RoboDK station: kr30 cnc 070419 1.rdk

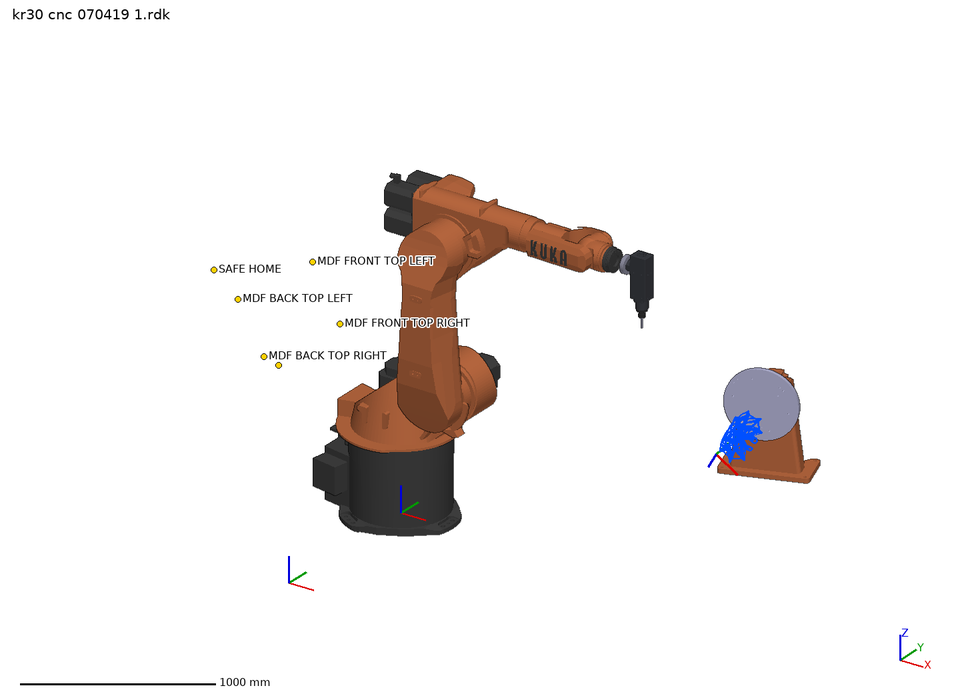
[picture v0: the station drawn from its stored meshes, robots at their saved joint values, targets as dots, program paths as lines]
Station kr30 cnc 070419 1. Poses are relative to the parent item; angles as X-Y-Z fixed-axis rotations.
  - frame GIGASHEEN 7th Axis Base at (0, 1000, 0) mm
    - robot KUKA KP1 MD250: 1 axes, payload 250 kg
        modified DH rows (alpha deg, a mm, theta deg, d mm): 0, 0, 0, 0
        base shift (1750, 1710, 820) mm, rotated rx 0 ry 90 rz -70 deg
        joint limits [-3600] to [3600]; home [0]; saved at [1487.65]
      - frame Reference Rhino at (0, -250, 250) mm
        - object RhinoPart at (0, 0, 0) mm
  - frame GIGASHEEN Base at (0, 2000, 0) mm
    - robot GIGASHEEN (model KUKA KR 30 HA): 6 axes, payload 30 kg, reach 2033 mm, repeatability 0.05 mm, weight 665 kg
        modified DH rows (alpha deg, a mm, theta deg, d mm): 0, 0, 0, 815; -90, 350, 0, 0; 0, 850, -90, 0; -90, 145, 0, 820; 90, 0, 0, 0; -90, 0, 180, 170
        joint limits [-185, -135, -120, -350, -119, -350] to [185, 35, 158, 350, 119, 350]; home [0, -90, 90, 0, 0, 0]; saved at [0, -90, 90, 0, 0, 0]
      - tool 1/2" End Mill TCP, TCP at (337.71, -2.2, 160.57) mm, rotated rx 0 ry 90 rz 0 deg, size 415.8 x 102 x 153.6 mm
    - target MDF BACK TOP LEFT (joint target) at (-335.18, -974.02, 1512.92) mm, rotated rx 85.17 ry 71.84 rz 47.05 deg; joints [27.716, -45.008, 102.25, 116.233, 75.695, -151.59, -681.46] of GIGASHEEN
    - target MDF FRONT TOP LEFT (joint target) at (-87.97, -665.25, 1668.52) mm, rotated rx 85.17 ry 71.84 rz 47.05 deg; joints [22.06, -21.631, 54.581, 104.768, 70.881, -126.376, -681.46] of GIGASHEEN
    - target MDF FRONT TOP RIGHT (joint target) at (4.03, -550.6, 1295.2) mm, rotated rx 85.17 ry 71.84 rz 47.05 deg; joints [10.053, -29.315, 70.245, 98.928, 81.917, -132.341, -681.46] of GIGASHEEN
    - target MDF BACK TOP RIGHT (joint target) at (-248.73, -867.72, 1165.36) mm, rotated rx 85.17 ry 71.84 rz 47.05 deg; joints [13.787, -50.344, 113.459, 104.66, 84.215, -154.683, -681.46] of GIGASHEEN
    - target MDF STOCK DEPTH (only use z axis value) (joint target) at (-166.67, -856.91, 1136.76) mm, rotated rx 85.17 ry 71.84 rz 47.05 deg; joints [11.502, -45.737, 110.222, 102.707, 85.519, -155.78, -681.46] of GIGASHEEN
    - target SAFE HOME (joint target) at (-1073.3, -134.71, 1136.76) mm, rotated rx 85.17 ry 71.84 rz 47.05 deg; joints [11.502, -69.45, 58.776, 88.861, 76.585, -79.989, -681.46] of GIGASHEEN
  - machining project RhinoPart Settings: rotZ(0) | rotX(90)*rotY(-155) | rotz(0)
  - program RhinoPart (1768 instructions, listed below)
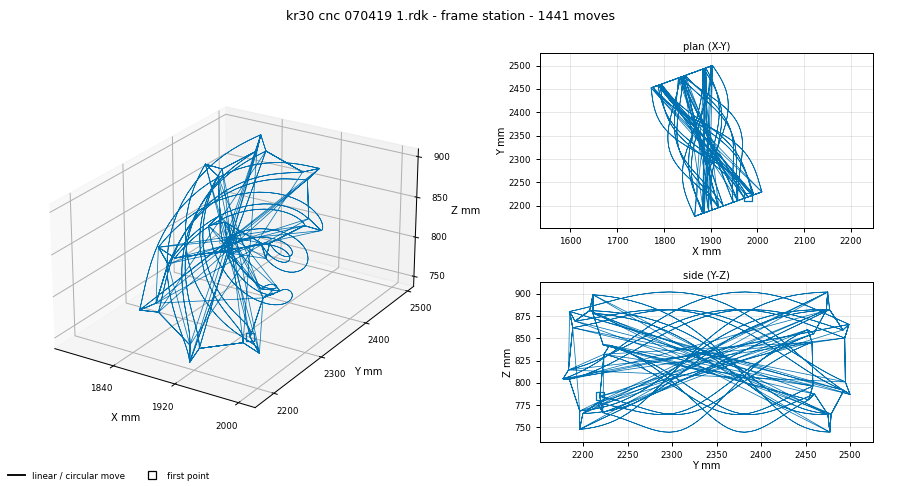
[picture p0: tool path of kr30 cnc 070419 1.rdk in frame station, 1441 of 1441 moves have a stored position in this frame; points joined in program order, loops and branches not executed]

--- program RhinoPart (robot GIGASHEEN) ---
  Set Ref.: Reference Rhino
  Set Tool: 1/2" End Mill TCP
  Show 1/2" End Mill TCP
  Set speed (1000.0 mm/s)
  MoveJ 1 to (58.93, 255.88, 290) mm, rotated rx -90 ry -25 rz 145.69 deg; joints [2.992, -45.858, 98.042, 40.619, -108.716, -6.951, -185.694]
  MoveL 2 to (58.93, 255.88, 290) mm, rotated rx -90 ry -25 rz 145.69 deg; joints [2.992, -45.858, 98.042, 40.619, -108.716, -6.951, -185.694]
  MoveL 3 to (58.93, 255.88, 290) mm, rotated rx -90 ry -25 rz 145.69 deg; joints [2.992, -45.858, 98.042, 40.619, -108.716, -6.951, -185.694]
  Set speed (60.0 mm/s)
  MoveL 4 to (37.11, 300.24, 290) mm, rotated rx -90 ry -25 rz -166.45 deg; joints [2.992, -46.004, 98.028, 40.584, -108.594, -7.061, -233.547]
  Set speed (1000.0 mm/s)
  MoveL 5 to (37.11, 300.24, 290) mm, rotated rx -90 ry -25 rz -166.45 deg; joints [2.992, -46.004, 98.028, 40.584, -108.594, -7.061, -233.547]
  Set speed (1000.0 mm/s)
  MoveL 6 to (-37.11, 208.63, 290) mm, rotated rx -90 ry -25 rz 8.11 deg; joints [2.992, -45.692, 98.056, 40.659, -108.852, -6.827, -408.107]
  MoveL 7 to (-37.11, 208.63, 290) mm, rotated rx -90 ry -25 rz 8.11 deg; joints [2.992, -45.692, 98.056, 40.659, -108.852, -6.827, -408.107]
  Set speed (60.0 mm/s)
  MoveL 8 to (-58.93, 252.99, 290) mm, rotated rx -90 ry -25 rz -42.9 deg; joints [2.992, -45.848, 98.043, 40.621, -108.724, -6.944, -357.096]
  Set speed (1000.0 mm/s)
  MoveL 9 to (-58.93, 252.99, 290) mm, rotated rx -90 ry -25 rz -42.9 deg; joints [2.992, -45.848, 98.043, 40.621, -108.724, -6.944, -357.096]
  Set speed (1000.0 mm/s)
  MoveL 10 to (21.11, 199.39, 290) mm, rotated rx -90 ry -25 rz 72.64 deg; joints [2.992, -45.658, 98.059, 40.667, -108.88, -6.802, -472.645]
  MoveL 11 to (21.11, 199.39, 290) mm, rotated rx -90 ry -25 rz 72.64 deg; joints [2.992, -45.658, 98.059, 40.667, -108.88, -6.802, -472.645]
  Set speed (60.0 mm/s)
  MoveL 12 to (34.79, 183.72, 290) mm, rotated rx -90 ry -25 rz 77.69 deg; joints [2.992, -46.56, 97.967, 40.451, -108.125, -7.483, -477.692]
  Set speed (1000.0 mm/s)
  MoveL 13 to (34.79, 183.72, 290) mm, rotated rx -90 ry -25 rz 77.69 deg; joints [2.992, -46.56, 97.967, 40.451, -108.125, -7.483, -477.692]
  Set speed (1000.0 mm/s)
  MoveL 14 to (21.11, 199.39, 290) mm, rotated rx -90 ry -25 rz 72.64 deg; joints [2.992, -45.658, 98.059, 40.667, -108.88, -6.802, -472.645]
  MoveL 15 to (21.11, 199.39, 290) mm, rotated rx -90 ry -25 rz 72.64 deg; joints [2.992, -45.658, 98.059, 40.667, -108.88, -6.802, -472.645]
  Set speed (60.0 mm/s)
  MoveL 16 to (-28.22, 202.67, 290) mm, rotated rx -90 ry -25 rz 19.2 deg; joints [2.992, -45.67, 98.058, 40.664, -108.87, -6.811, -419.196]
  Set speed (1000.0 mm/s)
  MoveL 17 to (-28.22, 202.67, 290) mm, rotated rx -90 ry -25 rz 19.2 deg; joints [2.992, -45.67, 98.058, 40.664, -108.87, -6.811, -419.196]
  Set speed (1000.0 mm/s)
  MoveL 18 to (-43.85, 188.95, 290) mm, rotated rx -90 ry -25 rz 14.31 deg; joints [2.992, -46.574, 97.966, 40.447, -108.114, -7.494, -414.314]
  MoveL 19 to (-43.85, 188.95, 290) mm, rotated rx -90 ry -25 rz 14.31 deg; joints [2.992, -46.574, 97.966, 40.447, -108.114, -7.494, -414.314]
  Set speed (60.0 mm/s)
  MoveL 20 to (-28.22, 202.67, 290) mm, rotated rx -90 ry -25 rz 19.2 deg; joints [2.992, -45.67, 98.058, 40.664, -108.87, -6.811, -419.196]
  Set speed (1000.0 mm/s)
  MoveL 21 to (-28.22, 202.67, 290) mm, rotated rx -90 ry -25 rz 19.2 deg; joints [2.992, -45.67, 98.058, 40.664, -108.87, -6.811, -419.196]
  Set speed (1000.0 mm/s)
  MoveL 22 to (-43.85, 188.95, 290) mm, rotated rx -90 ry -25 rz 14.31 deg; joints [2.992, -46.574, 97.966, 40.447, -108.114, -7.494, -414.314]
  MoveL 23 to (-43.85, 188.95, 290) mm, rotated rx -90 ry -25 rz 14.31 deg; joints [2.992, -46.574, 97.966, 40.447, -108.114, -7.494, -414.314]
  Set speed (60.0 mm/s)
  MoveL 24 to (-37.11, 208.63, 290) mm, rotated rx -90 ry -25 rz 8.11 deg; joints [2.992, -45.692, 98.056, 40.659, -108.852, -6.827, -408.107]
  Set speed (1000.0 mm/s)
  MoveL 25 to (-37.11, 208.63, 290) mm, rotated rx -90 ry -25 rz 8.11 deg; joints [2.992, -45.692, 98.056, 40.659, -108.852, -6.827, -408.107]
  Set speed (1000.0 mm/s)
  MoveL 26 to (-78.63, 259.66, 290) mm, rotated rx -90 ry -25 rz -47.01 deg; joints [2.992, -46.754, 97.943, 40.404, -107.959, -7.632, -352.994]
  MoveL 27 to (-78.63, 259.66, 290) mm, rotated rx -90 ry -25 rz -47.01 deg; joints [2.992, -46.754, 97.943, 40.404, -107.959, -7.632, -352.994]
  Set speed (60.0 mm/s)
  MoveL 28 to (-58.93, 252.99, 290) mm, rotated rx -90 ry -25 rz -42.9 deg; joints [2.992, -45.848, 98.043, 40.621, -108.724, -6.944, -357.096]
  Set speed (1000.0 mm/s)
  MoveL 29 to (-58.93, 252.99, 290) mm, rotated rx -90 ry -25 rz -42.9 deg; joints [2.992, -45.848, 98.043, 40.621, -108.724, -6.944, -357.096]
  Set speed (1000.0 mm/s)
  MoveL 30 to (-78.63, 259.66, 290) mm, rotated rx -90 ry -25 rz -47.01 deg; joints [2.992, -46.754, 97.943, 40.404, -107.959, -7.632, -352.994]
  MoveL 31 to (-78.63, 259.66, 290) mm, rotated rx -90 ry -25 rz -47.01 deg; joints [2.992, -46.754, 97.943, 40.404, -107.959, -7.632, -352.994]
  Set speed (60.0 mm/s)
  MoveL 32 to (-58.22, 263.67, 290) mm, rotated rx -90 ry -25 rz -53.21 deg; joints [2.992, -45.884, 98.039, 40.612, -108.694, -6.971, -346.787]
  Set speed (1000.0 mm/s)
  MoveL 33 to (-58.22, 263.67, 290) mm, rotated rx -90 ry -25 rz -53.21 deg; joints [2.992, -45.884, 98.039, 40.612, -108.694, -6.971, -346.787]
  Set speed (1000.0 mm/s)
  MoveL 34 to (-30.72, 304.75, 290) mm, rotated rx -90 ry -25 rz -100.71 deg; joints [2.992, -46.018, 98.027, 40.58, -108.582, -7.072, -299.294]
  MoveL 35 to (-30.72, 304.75, 290) mm, rotated rx -90 ry -25 rz -100.71 deg; joints [2.992, -46.018, 98.027, 40.58, -108.582, -7.072, -299.294]
  Set speed (60.0 mm/s)
  MoveL 36 to (-58.22, 263.67, 290) mm, rotated rx -90 ry -25 rz -53.21 deg; joints [2.992, -45.884, 98.039, 40.612, -108.694, -6.971, -346.787]
  Set speed (1000.0 mm/s)
  MoveL 37 to (-58.22, 263.67, 290) mm, rotated rx -90 ry -25 rz -53.21 deg; joints [2.992, -45.884, 98.039, 40.612, -108.694, -6.971, -346.787]
  Set speed (1000.0 mm/s)
  MoveL 38 to (-30.72, 304.75, 290) mm, rotated rx -90 ry -25 rz -100.71 deg; joints [2.992, -46.018, 98.027, 40.58, -108.582, -7.072, -299.294]
  MoveL 39 to (-30.72, 304.75, 290) mm, rotated rx -90 ry -25 rz -100.71 deg; joints [2.992, -46.018, 98.027, 40.58, -108.582, -7.072, -299.294]
  Set speed (60.0 mm/s)
  MoveL 40 to (-34.79, 325.15, 290) mm, rotated rx -90 ry -25 rz -105.16 deg; joints [2.992, -46.913, 97.922, 40.367, -107.822, -7.755, -294.84]
  Set speed (1000.0 mm/s)
  MoveL 41 to (-34.79, 325.15, 290) mm, rotated rx -90 ry -25 rz -105.16 deg; joints [2.992, -46.913, 97.922, 40.367, -107.822, -7.755, -294.84]
  Set speed (1000.0 mm/s)
  MoveL 42 to (-21.11, 309.47, 290) mm, rotated rx -90 ry -25 rz -110.46 deg; joints [2.992, -46.033, 98.025, 40.576, -108.57, -7.083, -289.544]
  MoveL 43 to (-21.11, 309.47, 290) mm, rotated rx -90 ry -25 rz -110.46 deg; joints [2.992, -46.033, 98.025, 40.576, -108.57, -7.083, -289.544]
  Set speed (60.0 mm/s)
  MoveL 44 to (-34.79, 325.15, 290) mm, rotated rx -90 ry -25 rz -105.16 deg; joints [2.992, -46.913, 97.922, 40.367, -107.822, -7.755, -294.84]
  Set speed (1000.0 mm/s)
  MoveL 45 to (-34.79, 325.15, 290) mm, rotated rx -90 ry -25 rz -105.16 deg; joints [2.992, -46.913, 97.922, 40.367, -107.822, -7.755, -294.84]
  Set speed (1000.0 mm/s)
  MoveL 46 to (-21.11, 309.47, 290) mm, rotated rx -90 ry -25 rz -110.46 deg; joints [2.992, -46.033, 98.025, 40.576, -108.57, -7.083, -289.544]
  MoveL 47 to (-21.11, 309.47, 290) mm, rotated rx -90 ry -25 rz -110.46 deg; joints [2.992, -46.033, 98.025, 40.576, -108.57, -7.083, -289.544]
  Set speed (60.0 mm/s)
  MoveL 48 to (28.22, 306.19, 290) mm, rotated rx -90 ry -25 rz -156.66 deg; joints [2.992, -46.023, 98.026, 40.579, -108.578, -7.075, -243.337]
  Set speed (1000.0 mm/s)
  MoveL 49 to (28.22, 306.19, 290) mm, rotated rx -90 ry -25 rz -156.66 deg; joints [2.992, -46.023, 98.026, 40.579, -108.578, -7.075, -243.337]
  Set speed (1000.0 mm/s)
  MoveL 50 to (43.85, 319.91, 290) mm, rotated rx -90 ry -25 rz -162.09 deg; joints [2.992, -46.901, 97.924, 40.37, -107.832, -7.745, -237.907]
  MoveL 51 to (43.85, 319.91, 290) mm, rotated rx -90 ry -25 rz -162.09 deg; joints [2.992, -46.901, 97.924, 40.37, -107.832, -7.745, -237.907]
  Set speed (60.0 mm/s)
  MoveL 52 to (28.22, 306.19, 290) mm, rotated rx -90 ry -25 rz -156.66 deg; joints [2.992, -46.023, 98.026, 40.579, -108.578, -7.075, -243.337]
  Set speed (1000.0 mm/s)
  MoveL 53 to (28.22, 306.19, 290) mm, rotated rx -90 ry -25 rz -156.66 deg; joints [2.992, -46.023, 98.026, 40.579, -108.578, -7.075, -243.337]
  Set speed (1000.0 mm/s)
  MoveL 54 to (43.85, 319.91, 290) mm, rotated rx -90 ry -25 rz -162.09 deg; joints [2.992, -46.901, 97.924, 40.37, -107.832, -7.745, -237.907]
  MoveL 55 to (43.85, 319.91, 290) mm, rotated rx -90 ry -25 rz -162.09 deg; joints [2.992, -46.901, 97.924, 40.37, -107.832, -7.745, -237.907]
  Set speed (60.0 mm/s)
  MoveL 56 to (37.11, 300.24, 290) mm, rotated rx -90 ry -25 rz -166.45 deg; joints [2.992, -46.004, 98.028, 40.584, -108.594, -7.061, -233.547]
  Set speed (1000.0 mm/s)
  MoveL 57 to (37.11, 300.24, 290) mm, rotated rx -90 ry -25 rz -166.45 deg; joints [2.992, -46.004, 98.028, 40.584, -108.594, -7.061, -233.547]
  Set speed (1000.0 mm/s)
  MoveL 58 to (78.63, 249.2, 290) mm, rotated rx -90 ry -25 rz 139.42 deg; joints [2.992, -46.728, 97.946, 40.411, -107.981, -7.612, -179.419]
  MoveL 59 to (78.63, 249.2, 290) mm, rotated rx -90 ry -25 rz 139.42 deg; joints [2.992, -46.728, 97.946, 40.411, -107.981, -7.612, -179.419]
  Set speed (60.0 mm/s)
  MoveL 60 to (58.93, 255.88, 290) mm, rotated rx -90 ry -25 rz 145.69 deg; joints [2.992, -45.858, 98.042, 40.619, -108.716, -6.951, -185.694]
  Set speed (1000.0 mm/s)
  MoveL 61 to (58.93, 255.88, 290) mm, rotated rx -90 ry -25 rz 145.69 deg; joints [2.992, -45.858, 98.042, 40.619, -108.716, -6.951, -185.694]
  Set speed (1000.0 mm/s)
  MoveL 62 to (78.63, 249.2, 290) mm, rotated rx -90 ry -25 rz 139.42 deg; joints [2.992, -46.728, 97.946, 40.411, -107.981, -7.612, -179.419]
  MoveL 63 to (78.63, 249.2, 290) mm, rotated rx -90 ry -25 rz 139.42 deg; joints [2.992, -46.728, 97.946, 40.411, -107.981, -7.612, -179.419]
  Set speed (60.0 mm/s)
  MoveL 64 to (58.22, 245.2, 290) mm, rotated rx -90 ry -25 rz 135.28 deg; joints [2.992, -45.821, 98.045, 40.627, -108.746, -6.924, -175.284]
  Set speed (1000.0 mm/s)
  MoveL 65 to (58.22, 245.2, 290) mm, rotated rx -90 ry -25 rz 135.28 deg; joints [2.992, -45.821, 98.045, 40.627, -108.746, -6.924, -175.284]
  Set speed (1000.0 mm/s)
  MoveL 66 to (30.72, 204.12, 290) mm, rotated rx -90 ry -25 rz 83.8 deg; joints [2.992, -45.676, 98.058, 40.663, -108.866, -6.815, -123.801]
  MoveL 67 to (30.72, 204.12, 290) mm, rotated rx -90 ry -25 rz 83.8 deg; joints [2.992, -45.676, 98.058, 40.663, -108.866, -6.815, -123.801]
  Set speed (60.0 mm/s)
  MoveL 68 to (58.22, 245.2, 290) mm, rotated rx -90 ry -25 rz 135.28 deg; joints [2.992, -45.821, 98.045, 40.627, -108.746, -6.924, -175.284]
  Set speed (1000.0 mm/s)
  MoveL 69 to (58.22, 245.2, 290) mm, rotated rx -90 ry -25 rz 135.28 deg; joints [2.992, -45.821, 98.045, 40.627, -108.746, -6.924, -175.284]
  Set speed (1000.0 mm/s)
  MoveL 70 to (30.72, 204.12, 290) mm, rotated rx -90 ry -25 rz 83.8 deg; joints [2.992, -45.676, 98.058, 40.663, -108.866, -6.815, -123.801]
  MoveL 71 to (30.72, 204.12, 290) mm, rotated rx -90 ry -25 rz 83.8 deg; joints [2.992, -45.676, 98.058, 40.663, -108.866, -6.815, -123.801]
  Set speed (60.0 mm/s)
  MoveL 72 to (34.79, 183.72, 290) mm, rotated rx -90 ry -25 rz 77.69 deg; joints [2.992, -46.56, 97.967, 40.451, -108.125, -7.483, -117.692]
  Set speed (1000.0 mm/s)
  MoveL 73 to (34.79, 183.72, 290) mm, rotated rx -90 ry -25 rz 77.69 deg; joints [2.992, -46.56, 97.967, 40.451, -108.125, -7.483, -117.692]
  Set speed (1000.0 mm/s)
  MoveL 74 to (-37.62, 299.82, 0) mm, rotated rx -90 ry -25 rz -92.94 deg; joints [-7.468, -50.311, 106.419, 34.538, -108.079, 0.675, 52.939]
  MoveL 75 to (-37.62, 299.82, 0) mm, rotated rx -90 ry -25 rz -92.94 deg; joints [-7.468, -50.311, 106.419, 34.538, -108.079, 0.675, 52.939]
  Set speed (60.0 mm/s)
  MoveL 76 to (10.16, 312.5, 0) mm, rotated rx -90 ry -25 rz -139.23 deg; joints [-7.468, -50.355, 106.415, 34.529, -108.039, 0.646, 99.233]
  Set speed (1000.0 mm/s)
  MoveL 77 to (10.16, 312.5, 0) mm, rotated rx -90 ry -25 rz -139.23 deg; joints [-7.468, -50.355, 106.415, 34.529, -108.039, 0.646, 99.233]
  Set speed (1000.0 mm/s)
  MoveL 78 to (-37.62, 299.82, 0) mm, rotated rx -90 ry -25 rz -92.94 deg; joints [-7.468, -50.311, 106.419, 34.538, -108.079, 0.675, 52.939]
  MoveL 79 to (-37.62, 299.82, 0) mm, rotated rx -90 ry -25 rz -92.94 deg; joints [-7.468, -50.311, 106.419, 34.538, -108.079, 0.675, 52.939]
  Set speed (60.0 mm/s)
  MoveL 80 to (-55.59, 310.29, 0) mm, rotated rx -90 ry -25 rz -87.32 deg; joints [-7.468, -51.259, 106.317, 34.349, -107.213, 0.052, 47.319]
  Set speed (1000.0 mm/s)
  MoveL 81 to (-55.59, 310.29, 0) mm, rotated rx -90 ry -25 rz -87.32 deg; joints [-7.468, -51.259, 106.317, 34.349, -107.213, 0.052, 47.319]
  Set speed (1000.0 mm/s)
  MoveL 82 to (-45.21, 292.27, 0) mm, rotated rx -90 ry -25 rz -83.07 deg; joints [-7.468, -50.285, 106.421, 34.543, -108.102, 0.692, 43.073]
  MoveL 83 to (-45.21, 292.27, 0) mm, rotated rx -90 ry -25 rz -83.07 deg; joints [-7.468, -50.285, 106.421, 34.543, -108.102, 0.692, 43.073]
  Set speed (60.0 mm/s)
  MoveL 84 to (-55.59, 310.29, 0) mm, rotated rx -90 ry -25 rz -87.32 deg; joints [-7.468, -51.259, 106.317, 34.349, -107.213, 0.052, 47.319]
  Set speed (1000.0 mm/s)
  MoveL 85 to (-55.59, 310.29, 0) mm, rotated rx -90 ry -25 rz -87.32 deg; joints [-7.468, -51.259, 106.317, 34.349, -107.213, 0.052, 47.319]
  Set speed (1000.0 mm/s)
  MoveL 86 to (-45.21, 292.27, 0) mm, rotated rx -90 ry -25 rz -83.07 deg; joints [-7.468, -50.285, 106.421, 34.543, -108.102, 0.692, 43.073]
  MoveL 87 to (-45.21, 292.27, 0) mm, rotated rx -90 ry -25 rz -83.07 deg; joints [-7.468, -50.285, 106.421, 34.543, -108.102, 0.692, 43.073]
  Set speed (60.0 mm/s)
  MoveL 88 to (-58.12, 244.54, 0) mm, rotated rx -90 ry -25 rz -34.64 deg; joints [-7.468, -50.113, 106.436, 34.578, -108.256, 0.804, -5.364]
  Set speed (1000.0 mm/s)
  MoveL 89 to (-58.12, 244.54, 0) mm, rotated rx -90 ry -25 rz -34.64 deg; joints [-7.468, -50.113, 106.436, 34.578, -108.256, 0.804, -5.364]
  Set speed (1000.0 mm/s)
  MoveL 90 to (-76.17, 234.21, 0) mm, rotated rx -90 ry -25 rz -28.29 deg; joints [-7.468, -51.057, 106.341, 34.389, -107.4, 0.186, -11.709]
  MoveL 91 to (-76.17, 234.21, 0) mm, rotated rx -90 ry -25 rz -28.29 deg; joints [-7.468, -51.057, 106.341, 34.389, -107.4, 0.186, -11.709]
  Set speed (60.0 mm/s)
  MoveL 92 to (-58.12, 244.54, 0) mm, rotated rx -90 ry -25 rz -34.64 deg; joints [-7.468, -50.113, 106.436, 34.578, -108.256, 0.804, -5.364]
  Set speed (1000.0 mm/s)
  MoveL 93 to (-58.12, 244.54, 0) mm, rotated rx -90 ry -25 rz -34.64 deg; joints [-7.468, -50.113, 106.436, 34.578, -108.256, 0.804, -5.364]
  Set speed (1000.0 mm/s)
  MoveL 94 to (-76.17, 234.21, 0) mm, rotated rx -90 ry -25 rz -28.29 deg; joints [-7.468, -51.057, 106.341, 34.389, -107.4, 0.186, -11.709]
  MoveL 95 to (-76.17, 234.21, 0) mm, rotated rx -90 ry -25 rz -28.29 deg; joints [-7.468, -51.057, 106.341, 34.389, -107.4, 0.186, -11.709]
  Set speed (60.0 mm/s)
  MoveL 96 to (-55.37, 234.2, 0) mm, rotated rx -90 ry -25 rz -24.07 deg; joints [-7.468, -50.074, 106.439, 34.586, -108.291, 0.829, -15.929]
  Set speed (1000.0 mm/s)
  MoveL 97 to (-55.37, 234.2, 0) mm, rotated rx -90 ry -25 rz -24.07 deg; joints [-7.468, -50.074, 106.439, 34.586, -108.291, 0.829, -15.929]
  Set speed (1000.0 mm/s)
  MoveL 98 to (-20.49, 199.16, 0) mm, rotated rx -90 ry -25 rz 28.05 deg; joints [-7.468, -49.938, 106.45, 34.613, -108.412, 0.917, -68.047]
  MoveL 99 to (-20.49, 199.16, 0) mm, rotated rx -90 ry -25 rz 28.05 deg; joints [-7.468, -49.938, 106.45, 34.613, -108.412, 0.917, -68.047]
  Set speed (60.0 mm/s)
  MoveL 100 to (-55.37, 234.2, 0) mm, rotated rx -90 ry -25 rz -24.07 deg; joints [-7.468, -50.074, 106.439, 34.586, -108.291, 0.829, -15.929]
  Set speed (1000.0 mm/s)
  MoveL 101 to (-55.37, 234.2, 0) mm, rotated rx -90 ry -25 rz -24.07 deg; joints [-7.468, -50.074, 106.439, 34.586, -108.291, 0.829, -15.929]
  Set speed (1000.0 mm/s)
  MoveL 102 to (-20.49, 199.16, 0) mm, rotated rx -90 ry -25 rz 28.05 deg; joints [-7.468, -49.938, 106.45, 34.613, -108.412, 0.917, -68.047]
  MoveL 103 to (-20.49, 199.16, 0) mm, rotated rx -90 ry -25 rz 28.05 deg; joints [-7.468, -49.938, 106.45, 34.613, -108.412, 0.917, -68.047]
  Set speed (60.0 mm/s)
  MoveL 104 to (-20.57, 178.36, 0) mm, rotated rx -90 ry -25 rz 33.98 deg; joints [-7.468, -50.9, 106.359, 34.42, -107.545, 0.29, -73.977]
  Set speed (1000.0 mm/s)
  MoveL 105 to (-20.57, 178.36, 0) mm, rotated rx -90 ry -25 rz 33.98 deg; joints [-7.468, -50.9, 106.359, 34.42, -107.545, 0.29, -73.977]
  Set speed (1000.0 mm/s)
  MoveL 106 to (-10.16, 196.36, 0) mm, rotated rx -90 ry -25 rz 39.27 deg; joints [-7.468, -49.927, 106.451, 34.616, -108.422, 0.924, -79.273]
  MoveL 107 to (-10.16, 196.36, 0) mm, rotated rx -90 ry -25 rz 39.27 deg; joints [-7.468, -49.927, 106.451, 34.616, -108.422, 0.924, -79.273]
  Set speed (60.0 mm/s)
  MoveL 108 to (-20.57, 178.36, 0) mm, rotated rx -90 ry -25 rz 33.98 deg; joints [-7.468, -50.9, 106.359, 34.42, -107.545, 0.29, -73.977]
  Set speed (1000.0 mm/s)
  MoveL 109 to (-20.57, 178.36, 0) mm, rotated rx -90 ry -25 rz 33.98 deg; joints [-7.468, -50.9, 106.359, 34.42, -107.545, 0.29, -73.977]
  Set speed (1000.0 mm/s)
  MoveL 110 to (-10.16, 196.36, 0) mm, rotated rx -90 ry -25 rz 39.27 deg; joints [-7.468, -49.927, 106.451, 34.616, -108.422, 0.924, -79.273]
  MoveL 111 to (-10.16, 196.36, 0) mm, rotated rx -90 ry -25 rz 39.27 deg; joints [-7.468, -49.927, 106.451, 34.616, -108.422, 0.924, -79.273]
  Set speed (60.0 mm/s)
  MoveL 112 to (37.62, 209.05, 0) mm, rotated rx -90 ry -25 rz 92.57 deg; joints [-7.468, -49.977, 106.447, 34.605, -108.377, 0.891, -132.574]
  Set speed (1000.0 mm/s)
  MoveL 113 to (37.62, 209.05, 0) mm, rotated rx -90 ry -25 rz 92.57 deg; joints [-7.468, -49.977, 106.447, 34.605, -108.377, 0.891, -132.574]
  Set speed (1000.0 mm/s)
  MoveL 114 to (55.59, 198.58, 0) mm, rotated rx -90 ry -25 rz 97.23 deg; joints [-7.468, -50.957, 106.353, 34.408, -107.492, 0.252, -137.234]
  MoveL 115 to (55.59, 198.58, 0) mm, rotated rx -90 ry -25 rz 97.23 deg; joints [-7.468, -50.957, 106.353, 34.408, -107.492, 0.252, -137.234]
  Set speed (60.0 mm/s)
  MoveL 116 to (37.62, 209.05, 0) mm, rotated rx -90 ry -25 rz 92.57 deg; joints [-7.468, -49.977, 106.447, 34.605, -108.377, 0.891, -132.574]
  Set speed (1000.0 mm/s)
  MoveL 117 to (37.62, 209.05, 0) mm, rotated rx -90 ry -25 rz 92.57 deg; joints [-7.468, -49.977, 106.447, 34.605, -108.377, 0.891, -132.574]
  Set speed (1000.0 mm/s)
  MoveL 118 to (55.59, 198.58, 0) mm, rotated rx -90 ry -25 rz 97.23 deg; joints [-7.468, -50.957, 106.353, 34.408, -107.492, 0.252, -137.234]
  MoveL 119 to (55.59, 198.58, 0) mm, rotated rx -90 ry -25 rz 97.23 deg; joints [-7.468, -50.957, 106.353, 34.408, -107.492, 0.252, -137.234]
  Set speed (60.0 mm/s)
  MoveL 120 to (45.21, 216.6, 0) mm, rotated rx -90 ry -25 rz 103.54 deg; joints [-7.468, -50.007, 106.445, 34.599, -108.351, 0.872, -143.543]
  Set speed (1000.0 mm/s)
  MoveL 121 to (45.21, 216.6, 0) mm, rotated rx -90 ry -25 rz 103.54 deg; joints [-7.468, -50.007, 106.445, 34.599, -108.351, 0.872, -143.543]
  Set speed (1000.0 mm/s)
  MoveL 122 to (58.12, 264.32, 0) mm, rotated rx -90 ry -25 rz 153.85 deg; joints [-7.468, -50.186, 106.43, 34.563, -108.191, 0.757, -193.845]
  MoveL 123 to (58.12, 264.32, 0) mm, rotated rx -90 ry -25 rz 153.85 deg; joints [-7.468, -50.186, 106.43, 34.563, -108.191, 0.757, -193.845]
  Set speed (60.0 mm/s)
  MoveL 124 to (45.21, 216.6, 0) mm, rotated rx -90 ry -25 rz 103.54 deg; joints [-7.468, -50.007, 106.445, 34.599, -108.351, 0.872, -143.543]
  Set speed (1000.0 mm/s)
  MoveL 125 to (45.21, 216.6, 0) mm, rotated rx -90 ry -25 rz 103.54 deg; joints [-7.468, -50.007, 106.445, 34.599, -108.351, 0.872, -143.543]
  Set speed (1000.0 mm/s)
  MoveL 126 to (58.12, 264.32, 0) mm, rotated rx -90 ry -25 rz 153.85 deg; joints [-7.468, -50.186, 106.43, 34.563, -108.191, 0.757, -193.845]
  MoveL 127 to (58.12, 264.32, 0) mm, rotated rx -90 ry -25 rz 153.85 deg; joints [-7.468, -50.186, 106.43, 34.563, -108.191, 0.757, -193.845]
  Set speed (60.0 mm/s)
  MoveL 128 to (76.17, 274.65, 0) mm, rotated rx -90 ry -25 rz 157.93 deg; joints [-7.468, -51.166, 106.328, 34.367, -107.299, 0.114, -197.935]
  Set speed (1000.0 mm/s)
  MoveL 129 to (76.17, 274.65, 0) mm, rotated rx -90 ry -25 rz 157.93 deg; joints [-7.468, -51.166, 106.328, 34.367, -107.299, 0.114, -197.935]
  Set speed (1000.0 mm/s)
  MoveL 130 to (55.37, 274.67, 0) mm, rotated rx -90 ry -25 rz 164.01 deg; joints [-7.468, -50.223, 106.427, 34.556, -108.158, 0.732, -204.014]
  MoveL 131 to (55.37, 274.67, 0) mm, rotated rx -90 ry -25 rz 164.01 deg; joints [-7.468, -50.223, 106.427, 34.556, -108.158, 0.732, -204.014]
  Set speed (60.0 mm/s)
  MoveL 132 to (76.17, 274.65, 0) mm, rotated rx -90 ry -25 rz 157.93 deg; joints [-7.468, -51.166, 106.328, 34.367, -107.299, 0.114, -197.935]
  Set speed (1000.0 mm/s)
  MoveL 133 to (76.17, 274.65, 0) mm, rotated rx -90 ry -25 rz 157.93 deg; joints [-7.468, -51.166, 106.328, 34.367, -107.299, 0.114, -197.935]
  Set speed (1000.0 mm/s)
  MoveL 134 to (55.37, 274.67, 0) mm, rotated rx -90 ry -25 rz 164.01 deg; joints [-7.468, -50.223, 106.427, 34.556, -108.158, 0.732, -204.014]
  MoveL 135 to (55.37, 274.67, 0) mm, rotated rx -90 ry -25 rz 164.01 deg; joints [-7.468, -50.223, 106.427, 34.556, -108.158, 0.732, -204.014]
  Set speed (60.0 mm/s)
  MoveL 136 to (20.49, 309.71, 0) mm, rotated rx -90 ry -25 rz -148.94 deg; joints [-7.468, -50.346, 106.416, 34.531, -108.048, 0.653, -251.057]
  Set speed (1000.0 mm/s)
  MoveL 137 to (20.49, 309.71, 0) mm, rotated rx -90 ry -25 rz -148.94 deg; joints [-7.468, -50.346, 106.416, 34.531, -108.048, 0.653, -251.057]
  Set speed (1000.0 mm/s)
  MoveL 138 to (20.57, 330.51, 0) mm, rotated rx -90 ry -25 rz -144.34 deg; joints [-7.468, -51.311, 106.31, 34.338, -107.164, 0.017, -255.665]
  MoveL 139 to (20.57, 330.51, 0) mm, rotated rx -90 ry -25 rz -144.34 deg; joints [-7.468, -51.311, 106.31, 34.338, -107.164, 0.017, -255.665]
  Set speed (60.0 mm/s)
  MoveL 140 to (20.49, 309.71, 0) mm, rotated rx -90 ry -25 rz -148.94 deg; joints [-7.468, -50.346, 106.416, 34.531, -108.048, 0.653, -251.057]
  Set speed (1000.0 mm/s)
  MoveL 141 to (20.49, 309.71, 0) mm, rotated rx -90 ry -25 rz -148.94 deg; joints [-7.468, -50.346, 106.416, 34.531, -108.048, 0.653, -251.057]
  Set speed (1000.0 mm/s)
  MoveL 142 to (20.57, 330.51, 0) mm, rotated rx -90 ry -25 rz -144.34 deg; joints [-7.468, -51.311, 106.31, 34.338, -107.164, 0.017, -255.665]
  MoveL 143 to (20.57, 330.51, 0) mm, rotated rx -90 ry -25 rz -144.34 deg; joints [-7.468, -51.311, 106.31, 34.338, -107.164, 0.017, -255.665]
  Set speed (60.0 mm/s)
  MoveL 144 to (10.16, 312.5, 0) mm, rotated rx -90 ry -25 rz -139.23 deg; joints [-7.468, -50.355, 106.415, 34.529, -108.039, 0.646, -260.767]
  Set speed (1000.0 mm/s)
  MoveL 145 to (10.16, 312.5, 0) mm, rotated rx -90 ry -25 rz -139.23 deg; joints [-7.468, -50.355, 106.415, 34.529, -108.039, 0.646, -260.767]
  Set speed (1000.0 mm/s)
  MoveL 146 to (-37.62, 299.82, 0) mm, rotated rx -90 ry -25 rz -92.94 deg; joints [-7.468, -50.311, 106.419, 34.538, -108.079, 0.675, -307.061]
  MoveL 147 to (-37.62, 299.82, 0) mm, rotated rx -90 ry -25 rz -92.94 deg; joints [-7.468, -50.311, 106.419, 34.538, -108.079, 0.675, -307.061]
  Set speed (60.0 mm/s)
  MoveL 148 to (-40.85, 296.93, 10) mm, rotated rx -90 ry -25 rz -88.96 deg; joints [-7.088, -50.198, 106.219, 34.78, -108.128, 0.44, -311.039]
  MoveL 149 to (-44.15, 293.5, 20) mm, rotated rx -90 ry -25 rz -84.58 deg; joints [-6.709, -50.079, 106.012, 35.02, -108.177, 0.204, -315.425]
  MoveL 150 to (-47.39, 289.5, 30) mm, rotated rx -90 ry -25 rz -79.81 deg; joints [-6.332, -49.955, 105.8, 35.259, -108.227, -0.032, -320.19]
  MoveL 151 to (-50.45, 284.92, 40) mm, rotated rx -90 ry -25 rz -74.69 deg; joints [-5.956, -49.826, 105.582, 35.496, -108.277, -0.268, -325.308]
  MoveL 152 to (-53.21, 279.8, 50) mm, rotated rx -90 ry -25 rz -69.25 deg; joints [-5.581, -49.692, 105.357, 35.732, -108.326, -0.504, -330.751]
  MoveL 153 to (-55.55, 274.16, 60) mm, rotated rx -90 ry -25 rz -63.51 deg; joints [-5.207, -49.552, 105.127, 35.966, -108.376, -0.74, -336.493]
  MoveL 154 to (-57.35, 268.08, 70) mm, rotated rx -90 ry -25 rz -57.49 deg; joints [-4.834, -49.408, 104.89, 36.198, -108.425, -0.977, -342.507]
  MoveL 155 to (-58.51, 261.62, 80) mm, rotated rx -90 ry -25 rz -51.24 deg; joints [-4.463, -49.259, 104.647, 36.429, -108.474, -1.215, -348.765]
  MoveL 156 to (-58.95, 254.91, 90) mm, rotated rx -90 ry -25 rz -44.76 deg; joints [-4.093, -49.106, 104.398, 36.657, -108.522, -1.454, -355.24]
  MoveL 157 to (-58.6, 248.05, 100) mm, rotated rx -90 ry -25 rz -38.1 deg; joints [-3.725, -48.95, 104.143, 36.884, -108.569, -1.693, -361.902]
  MoveL 158 to (-57.44, 241.19, 110) mm, rotated rx -90 ry -25 rz -31.28 deg; joints [-3.358, -48.79, 103.881, 37.108, -108.614, -1.935, -368.721]
  MoveL 159 to (-55.46, 234.45, 120) mm, rotated rx -90 ry -25 rz -24.34 deg; joints [-2.992, -48.627, 103.613, 37.33, -108.658, -2.178, -375.664]
  MoveL 160 to (-52.68, 227.97, 130) mm, rotated rx -90 ry -25 rz -17.3 deg; joints [-2.628, -48.462, 103.339, 37.55, -108.698, -2.423, -382.696]
  MoveL 161 to (-49.15, 221.88, 140) mm, rotated rx -90 ry -25 rz -10.22 deg; joints [-2.265, -48.294, 103.059, 37.767, -108.736, -2.671, -389.78]
  MoveL 162 to (-44.94, 216.28, 150) mm, rotated rx -90 ry -25 rz -3.12 deg; joints [-1.904, -48.126, 102.771, 37.981, -108.771, -2.922, -396.877]
  MoveL 163 to (-40.17, 211.29, 160) mm, rotated rx -90 ry -25 rz 3.94 deg; joints [-1.544, -47.956, 102.478, 38.192, -108.802, -3.176, -403.944]
  MoveL 164 to (-34.94, 206.95, 170) mm, rotated rx -90 ry -25 rz 10.94 deg; joints [-1.185, -47.786, 102.178, 38.401, -108.829, -3.434, -410.939]
  MoveL 165 to (-29.38, 203.32, 180) mm, rotated rx -90 ry -25 rz 17.81 deg; joints [-0.828, -47.615, 101.871, 38.606, -108.852, -3.696, -417.814]
  MoveL 166 to (-23.62, 200.42, 190) mm, rotated rx -90 ry -25 rz 24.52 deg; joints [-0.473, -47.444, 101.557, 38.809, -108.871, -3.961, -424.525]
  MoveL 167 to (-17.8, 198.23, 200) mm, rotated rx -90 ry -25 rz 31.02 deg; joints [-0.119, -47.272, 101.237, 39.008, -108.886, -4.23, -431.023]
  MoveL 168 to (-12.04, 196.73, 210) mm, rotated rx -90 ry -25 rz 37.26 deg; joints [0.233, -47.1, 100.911, 39.204, -108.897, -4.503, -437.262]
  MoveL 169 to (-6.46, 195.84, 220) mm, rotated rx -90 ry -25 rz 43.2 deg; joints [0.584, -46.927, 100.577, 39.397, -108.905, -4.78, -443.197]
  MoveL 170 to (-1.16, 195.49, 230) mm, rotated rx -90 ry -25 rz 48.78 deg; joints [0.933, -46.752, 100.237, 39.587, -108.909, -5.06, -448.782]
  MoveL 171 to (3.78, 195.6, 240) mm, rotated rx -90 ry -25 rz 53.97 deg; joints [1.28, -46.576, 99.891, 39.774, -108.91, -5.344, -453.974]
  MoveL 172 to (8.28, 196.07, 250) mm, rotated rx -90 ry -25 rz 58.73 deg; joints [1.626, -46.398, 99.538, 39.958, -108.908, -5.631, -458.733]
  MoveL 173 to (12.3, 196.78, 260) mm, rotated rx -90 ry -25 rz 63.02 deg; joints [1.97, -46.218, 99.178, 40.139, -108.904, -5.92, -463.017]
  MoveL 174 to (15.8, 197.64, 270) mm, rotated rx -90 ry -25 rz 66.79 deg; joints [2.312, -46.035, 98.812, 40.318, -108.898, -6.212, -466.788]
  MoveL 175 to (18.74, 198.54, 280) mm, rotated rx -90 ry -25 rz 70.01 deg; joints [2.653, -45.848, 98.439, 40.494, -108.89, -6.506, -470.01]
  MoveL 176 to (21.11, 199.39, 290) mm, rotated rx -90 ry -25 rz 72.64 deg; joints [2.992, -45.658, 98.059, 40.667, -108.88, -6.802, -472.645]
  Set speed (1000.0 mm/s)
  MoveL 177 to (21.11, 199.39, 290) mm, rotated rx -90 ry -25 rz 72.64 deg; joints [2.992, -45.658, 98.059, 40.667, -108.88, -6.802, -472.645]
  Set speed (1000.0 mm/s)
  MoveL 178 to (10.16, 312.5, 0) mm, rotated rx -90 ry -25 rz -139.23 deg; joints [-7.468, -50.355, 106.415, 34.529, -108.039, 0.646, -620.767]
  MoveL 179 to (10.16, 312.5, 0) mm, rotated rx -90 ry -25 rz -139.23 deg; joints [-7.468, -50.355, 106.415, 34.529, -108.039, 0.646, -620.767]
  Set speed (60.0 mm/s)
  MoveL 180 to (-37.62, 299.82, 0) mm, rotated rx -90 ry -25 rz -92.94 deg; joints [-7.468, -50.311, 106.419, 34.538, -108.079, 0.675, -667.061]
  Set speed (1000.0 mm/s)
  MoveL 181 to (-37.62, 299.82, 0) mm, rotated rx -90 ry -25 rz -92.94 deg; joints [-7.468, -50.311, 106.419, 34.538, -108.079, 0.675, -667.061]
  Set speed (1000.0 mm/s)
  MoveL 182 to (-28.22, 202.67, 290) mm, rotated rx -90 ry -25 rz 19.2 deg; joints [2.992, -45.67, 98.058, 40.664, -108.87, -6.811, -779.196]
  MoveL 183 to (-28.22, 202.67, 290) mm, rotated rx -90 ry -25 rz 19.2 deg; joints [2.992, -45.67, 98.058, 40.664, -108.87, -6.811, -779.196]
  Set speed (60.0 mm/s)
  MoveL 184 to (21.11, 199.39, 290) mm, rotated rx -90 ry -25 rz 72.64 deg; joints [2.992, -45.658, 98.059, 40.667, -108.88, -6.802, -832.645]
  Set speed (1000.0 mm/s)
  MoveL 185 to (21.11, 199.39, 290) mm, rotated rx -90 ry -25 rz 72.64 deg; joints [2.992, -45.658, 98.059, 40.667, -108.88, -6.802, -832.645]
  Set speed (1000.0 mm/s)
  MoveL 186 to (-28.22, 202.67, 290) mm, rotated rx -90 ry -25 rz 19.2 deg; joints [2.992, -45.67, 98.058, 40.664, -108.87, -6.811, -779.196]
  MoveL 187 to (-28.22, 202.67, 290) mm, rotated rx -90 ry -25 rz 19.2 deg; joints [2.992, -45.67, 98.058, 40.664, -108.87, -6.811, -779.196]
  Set speed (60.0 mm/s)
  MoveL 188 to (-30.4, 203.93, 280) mm, rotated rx -90 ry -25 rz 16.58 deg; joints [2.653, -45.868, 98.437, 40.489, -108.873, -6.521, -776.579]
  MoveL 189 to (-33, 205.58, 270) mm, rotated rx -90 ry -25 rz 13.39 deg; joints [2.312, -46.064, 98.809, 40.311, -108.874, -6.234, -773.391]
  MoveL 190 to (-35.92, 207.69, 260) mm, rotated rx -90 ry -25 rz 9.67 deg; joints [1.97, -46.258, 99.175, 40.13, -108.871, -5.95, -769.674]
  MoveL 191 to (-39.07, 210.28, 250) mm, rotated rx -90 ry -25 rz 5.47 deg; joints [1.626, -46.451, 99.533, 39.946, -108.865, -5.669, -765.473]
  MoveL 192 to (-42.34, 213.41, 240) mm, rotated rx -90 ry -25 rz 0.83 deg; joints [1.28, -46.642, 99.885, 39.758, -108.855, -5.392, -760.831]
  MoveL 193 to (-45.62, 217.1, 230) mm, rotated rx -90 ry -25 rz -4.21 deg; joints [0.933, -46.832, 100.231, 39.568, -108.842, -5.119, -755.794]
  MoveL 194 to (-48.8, 221.36, 220) mm, rotated rx -90 ry -25 rz -9.59 deg; joints [0.584, -47.021, 100.57, 39.375, -108.826, -4.849, -750.406]
  MoveL 195 to (-51.74, 226.19, 210) mm, rotated rx -90 ry -25 rz -15.29 deg; joints [0.233, -47.209, 100.902, 39.178, -108.806, -4.582, -744.713]
  MoveL 196 to (-54.33, 231.55, 200) mm, rotated rx -90 ry -25 rz -21.24 deg; joints [-0.119, -47.395, 101.227, 38.979, -108.783, -4.319, -738.758]
  MoveL 197 to (-56.44, 237.4, 190) mm, rotated rx -90 ry -25 rz -27.41 deg; joints [-0.473, -47.58, 101.546, 38.777, -108.756, -4.059, -732.587]
  MoveL 198 to (-57.96, 243.66, 180) mm, rotated rx -90 ry -25 rz -33.76 deg; joints [-0.828, -47.763, 101.858, 38.572, -108.727, -3.801, -726.24]
  MoveL 199 to (-58.8, 250.25, 170) mm, rotated rx -90 ry -25 rz -40.24 deg; joints [-1.185, -47.944, 102.164, 38.365, -108.694, -3.547, -719.76]
  MoveL 200 to (-58.89, 257.04, 160) mm, rotated rx -90 ry -25 rz -46.82 deg; joints [-1.544, -48.123, 102.464, 38.154, -108.66, -3.294, -713.183]
  MoveL 201 to (-58.18, 263.92, 150) mm, rotated rx -90 ry -25 rz -53.45 deg; joints [-1.904, -48.298, 102.757, 37.942, -108.623, -3.043, -706.549]
  MoveL 202 to (-56.65, 270.74, 140) mm, rotated rx -90 ry -25 rz -60.11 deg; joints [-2.265, -48.47, 103.043, 37.727, -108.585, -2.794, -699.89]
  MoveL 203 to (-54.3, 277.38, 130) mm, rotated rx -90 ry -25 rz -66.76 deg; joints [-2.628, -48.638, 103.324, 37.51, -108.546, -2.546, -693.241]
  MoveL 204 to (-51.17, 283.7, 120) mm, rotated rx -90 ry -25 rz -73.37 deg; joints [-2.992, -48.802, 103.598, 37.291, -108.506, -2.299, -686.632]
  MoveL 205 to (-47.33, 289.58, 110) mm, rotated rx -90 ry -25 rz -79.91 deg; joints [-3.358, -48.961, 103.866, 37.07, -108.466, -2.053, -680.094]
  MoveL 206 to (-42.85, 294.92, 100) mm, rotated rx -90 ry -25 rz -86.35 deg; joints [-3.725, -49.114, 104.128, 36.848, -108.426, -1.807, -673.654]
  MoveL 207 to (-37.86, 299.62, 90) mm, rotated rx -90 ry -25 rz -92.66 deg; joints [-4.093, -49.263, 104.384, 36.623, -108.386, -1.561, -667.341]
  MoveL 208 to (-32.46, 303.64, 80) mm, rotated rx -90 ry -25 rz -98.82 deg; joints [-4.463, -49.406, 104.634, 36.397, -108.346, -1.315, -661.181]
  MoveL 209 to (-26.8, 306.94, 70) mm, rotated rx -90 ry -25 rz -104.8 deg; joints [-4.834, -49.543, 104.878, 36.169, -108.307, -1.069, -655.202]
  MoveL 210 to (-21, 309.52, 60) mm, rotated rx -90 ry -25 rz -110.57 deg; joints [-5.207, -49.675, 105.115, 35.94, -108.268, -0.823, -649.431]
  MoveL 211 to (-15.19, 311.39, 50) mm, rotated rx -90 ry -25 rz -116.1 deg; joints [-5.581, -49.801, 105.347, 35.709, -108.23, -0.577, -643.896]
  MoveL 212 to (-9.5, 312.61, 40) mm, rotated rx -90 ry -25 rz -121.38 deg; joints [-5.956, -49.921, 105.573, 35.476, -108.192, -0.331, -638.624]
  MoveL 213 to (-4.03, 313.25, 30) mm, rotated rx -90 ry -25 rz -126.35 deg; joints [-6.332, -50.037, 105.793, 35.242, -108.154, -0.086, -633.645]
  MoveL 214 to (1.12, 313.37, 20) mm, rotated rx -90 ry -25 rz -131.01 deg; joints [-6.709, -50.147, 106.006, 35.006, -108.116, 0.159, -628.989]
  MoveL 215 to (5.87, 313.09, 10) mm, rotated rx -90 ry -25 rz -135.31 deg; joints [-7.088, -50.253, 106.214, 34.768, -108.078, 0.403, -624.685]
  MoveL 216 to (10.16, 312.5, 0) mm, rotated rx -90 ry -25 rz -139.23 deg; joints [-7.468, -50.355, 106.415, 34.529, -108.039, 0.646, -620.767]
  Set speed (1000.0 mm/s)
  MoveL 217 to (10.16, 312.5, 0) mm, rotated rx -90 ry -25 rz -139.23 deg; joints [-7.468, -50.355, 106.415, 34.529, -108.039, 0.646, -620.767]
  Set speed (1000.0 mm/s)
  MoveL 218 to (-37.62, 299.82, 0) mm, rotated rx -90 ry -25 rz -92.94 deg; joints [-7.468, -50.311, 106.419, 34.538, -108.079, 0.675, -667.061]
  MoveL 219 to (-37.62, 299.82, 0) mm, rotated rx -90 ry -25 rz -92.94 deg; joints [-7.468, -50.311, 106.419, 34.538, -108.079, 0.675, -667.061]
  Set speed (60.0 mm/s)
  MoveL 220 to (-40.85, 296.93, 10) mm, rotated rx -90 ry -25 rz -88.96 deg; joints [-7.088, -50.198, 106.219, 34.78, -108.128, 0.44, -671.039]
  MoveL 221 to (-44.15, 293.5, 20) mm, rotated rx -90 ry -25 rz -84.58 deg; joints [-6.709, -50.079, 106.012, 35.02, -108.177, 0.204, -675.425]
  MoveL 222 to (-47.39, 289.5, 30) mm, rotated rx -90 ry -25 rz -79.81 deg; joints [-6.332, -49.955, 105.8, 35.259, -108.227, -0.032, -680.19]
  MoveL 223 to (-50.45, 284.92, 40) mm, rotated rx -90 ry -25 rz -74.69 deg; joints [-5.956, -49.826, 105.582, 35.496, -108.277, -0.268, -685.308]
  MoveL 224 to (-53.21, 279.8, 50) mm, rotated rx -90 ry -25 rz -69.25 deg; joints [-5.581, -49.692, 105.357, 35.732, -108.326, -0.504, -690.751]
  MoveL 225 to (-55.55, 274.16, 60) mm, rotated rx -90 ry -25 rz -63.51 deg; joints [-5.207, -49.552, 105.127, 35.966, -108.376, -0.74, -696.493]
  MoveL 226 to (-57.35, 268.08, 70) mm, rotated rx -90 ry -25 rz -57.49 deg; joints [-4.834, -49.408, 104.89, 36.198, -108.425, -0.977, -702.507]
  MoveL 227 to (-58.51, 261.62, 80) mm, rotated rx -90 ry -25 rz -51.24 deg; joints [-4.463, -49.259, 104.647, 36.429, -108.474, -1.215, -708.765]
  MoveL 228 to (-58.95, 254.91, 90) mm, rotated rx -90 ry -25 rz -44.76 deg; joints [-4.093, -49.106, 104.398, 36.657, -108.522, -1.454, -715.24]
  MoveL 229 to (-58.6, 248.05, 100) mm, rotated rx -90 ry -25 rz -38.1 deg; joints [-3.725, -48.95, 104.143, 36.884, -108.569, -1.693, -721.902]
  MoveL 230 to (-57.44, 241.19, 110) mm, rotated rx -90 ry -25 rz -31.28 deg; joints [-3.358, -48.79, 103.881, 37.108, -108.614, -1.935, -728.721]
  MoveL 231 to (-55.46, 234.45, 120) mm, rotated rx -90 ry -25 rz -24.34 deg; joints [-2.992, -48.627, 103.613, 37.33, -108.658, -2.178, -735.664]
  MoveL 232 to (-52.68, 227.97, 130) mm, rotated rx -90 ry -25 rz -17.3 deg; joints [-2.628, -48.462, 103.339, 37.55, -108.698, -2.423, -742.696]
  MoveL 233 to (-49.15, 221.88, 140) mm, rotated rx -90 ry -25 rz -10.22 deg; joints [-2.265, -48.294, 103.059, 37.767, -108.736, -2.671, -749.78]
  MoveL 234 to (-44.94, 216.28, 150) mm, rotated rx -90 ry -25 rz -3.12 deg; joints [-1.904, -48.126, 102.771, 37.981, -108.771, -2.922, -756.877]
  MoveL 235 to (-40.17, 211.29, 160) mm, rotated rx -90 ry -25 rz 3.94 deg; joints [-1.544, -47.956, 102.478, 38.192, -108.802, -3.176, -763.944]
  MoveL 236 to (-34.94, 206.95, 170) mm, rotated rx -90 ry -25 rz 10.94 deg; joints [-1.185, -47.786, 102.178, 38.401, -108.829, -3.434, -770.939]
  MoveL 237 to (-29.38, 203.32, 180) mm, rotated rx -90 ry -25 rz 17.81 deg; joints [-0.828, -47.615, 101.871, 38.606, -108.852, -3.696, -777.814]
  MoveL 238 to (-23.62, 200.42, 190) mm, rotated rx -90 ry -25 rz 24.52 deg; joints [-0.473, -47.444, 101.557, 38.809, -108.871, -3.961, -784.525]
  MoveL 239 to (-17.8, 198.23, 200) mm, rotated rx -90 ry -25 rz 31.02 deg; joints [-0.119, -47.272, 101.237, 39.008, -108.886, -4.23, -791.023]
  MoveL 240 to (-12.04, 196.73, 210) mm, rotated rx -90 ry -25 rz 37.26 deg; joints [0.233, -47.1, 100.911, 39.204, -108.897, -4.503, -797.262]
  MoveL 241 to (-6.46, 195.84, 220) mm, rotated rx -90 ry -25 rz 43.2 deg; joints [0.584, -46.927, 100.577, 39.397, -108.905, -4.78, -803.197]
  MoveL 242 to (-1.16, 195.49, 230) mm, rotated rx -90 ry -25 rz 48.78 deg; joints [0.933, -46.752, 100.237, 39.587, -108.909, -5.06, -808.782]
  MoveL 243 to (3.78, 195.6, 240) mm, rotated rx -90 ry -25 rz 53.97 deg; joints [1.28, -46.576, 99.891, 39.774, -108.91, -5.344, -813.974]
  MoveL 244 to (8.28, 196.07, 250) mm, rotated rx -90 ry -25 rz 58.73 deg; joints [1.626, -46.398, 99.538, 39.958, -108.908, -5.631, -818.733]
  MoveL 245 to (12.3, 196.78, 260) mm, rotated rx -90 ry -25 rz 63.02 deg; joints [1.97, -46.218, 99.178, 40.139, -108.904, -5.92, -823.017]
  MoveL 246 to (15.8, 197.64, 270) mm, rotated rx -90 ry -25 rz 66.79 deg; joints [2.312, -46.035, 98.812, 40.318, -108.898, -6.212, -826.788]
  MoveL 247 to (18.74, 198.54, 280) mm, rotated rx -90 ry -25 rz 70.01 deg; joints [2.653, -45.848, 98.439, 40.494, -108.89, -6.506, -830.01]
  MoveL 248 to (21.11, 199.39, 290) mm, rotated rx -90 ry -25 rz 72.64 deg; joints [2.992, -45.658, 98.059, 40.667, -108.88, -6.802, -832.645]
  Set speed (1000.0 mm/s)
  MoveL 249 to (21.11, 199.39, 290) mm, rotated rx -90 ry -25 rz 72.64 deg; joints [2.992, -45.658, 98.059, 40.667, -108.88, -6.802, -832.645]
  Set speed (1000.0 mm/s)
  MoveL 250 to (34.79, 183.72, 290) mm, rotated rx -90 ry -25 rz 77.69 deg; joints [2.992, -46.56, 97.967, 40.451, -108.125, -7.483, -837.692]
  MoveL 251 to (34.79, 183.72, 290) mm, rotated rx -90 ry -25 rz 77.69 deg; joints [2.992, -46.56, 97.967, 40.451, -108.125, -7.483, -837.692]
  Set speed (60.0 mm/s)
  MoveL 252 to (21.11, 199.39, 290) mm, rotated rx -90 ry -25 rz 72.64 deg; joints [2.992, -45.658, 98.059, 40.667, -108.88, -6.802, -832.645]
  Set speed (1000.0 mm/s)
  MoveL 253 to (21.11, 199.39, 290) mm, rotated rx -90 ry -25 rz 72.64 deg; joints [2.992, -45.658, 98.059, 40.667, -108.88, -6.802, -832.645]
  Set speed (1000.0 mm/s)
  MoveL 254 to (-55.59, 310.29, 0) mm, rotated rx -90 ry -25 rz -87.32 deg; joints [-7.468, -51.259, 106.317, 34.349, -107.213, 0.052, -672.681]
  MoveL 255 to (-55.59, 310.29, 0) mm, rotated rx -90 ry -25 rz -87.32 deg; joints [-7.468, -51.259, 106.317, 34.349, -107.213, 0.052, -672.681]
  Set speed (60.0 mm/s)
  MoveL 256 to (-37.62, 299.82, 0) mm, rotated rx -90 ry -25 rz -92.94 deg; joints [-7.468, -50.311, 106.419, 34.538, -108.079, 0.675, -667.061]
  Set speed (1000.0 mm/s)
  MoveL 257 to (-37.62, 299.82, 0) mm, rotated rx -90 ry -25 rz -92.94 deg; joints [-7.468, -50.311, 106.419, 34.538, -108.079, 0.675, -667.061]
  Set speed (1000.0 mm/s)
  MoveL 258 to (34.79, 183.72, 290) mm, rotated rx -90 ry -25 rz 77.69 deg; joints [2.992, -46.56, 97.967, 40.451, -108.125, -7.483, -837.692]
  MoveL 259 to (34.79, 183.72, 290) mm, rotated rx -90 ry -25 rz 77.69 deg; joints [2.992, -46.56, 97.967, 40.451, -108.125, -7.483, -837.692]
  Set speed (60.0 mm/s)
  MoveL 260 to (31.73, 182.3, 280) mm, rotated rx -90 ry -25 rz 75.11 deg; joints [2.653, -46.752, 98.347, 40.278, -108.131, -7.186, -835.112]
  MoveL 261 to (27.92, 180.74, 270) mm, rotated rx -90 ry -25 rz 71.96 deg; joints [2.312, -46.941, 98.72, 40.102, -108.136, -6.891, -831.958]
  MoveL 262 to (23.38, 179.17, 260) mm, rotated rx -90 ry -25 rz 68.27 deg; joints [1.97, -47.126, 99.087, 39.924, -108.139, -6.598, -828.265]
  MoveL 263 to (18.11, 177.74, 250) mm, rotated rx -90 ry -25 rz 64.07 deg; joints [1.626, -47.308, 99.447, 39.743, -108.14, -6.307, -824.071]
  MoveL 264 to (12.17, 176.57, 240) mm, rotated rx -90 ry -25 rz 59.41 deg; joints [1.28, -47.487, 99.8, 39.56, -108.139, -6.019, -819.412]
  MoveL 265 to (5.61, 175.83, 230) mm, rotated rx -90 ry -25 rz 54.33 deg; joints [0.933, -47.665, 100.147, 39.373, -108.135, -5.733, -814.325]
  MoveL 266 to (-1.49, 175.64, 220) mm, rotated rx -90 ry -25 rz 48.85 deg; joints [0.584, -47.84, 100.487, 39.184, -108.128, -5.451, -808.851]
  MoveL 267 to (-9.03, 176.15, 210) mm, rotated rx -90 ry -25 rz 43.03 deg; joints [0.233, -48.014, 100.82, 38.992, -108.118, -5.172, -803.03]
  MoveL 268 to (-16.88, 177.46, 200) mm, rotated rx -90 ry -25 rz 36.9 deg; joints [-0.119, -48.187, 101.147, 38.797, -108.104, -4.896, -796.902]
  MoveL 269 to (-24.89, 179.66, 190) mm, rotated rx -90 ry -25 rz 30.51 deg; joints [-0.473, -48.36, 101.467, 38.598, -108.086, -4.624, -790.512]
  MoveL 270 to (-32.91, 182.83, 180) mm, rotated rx -90 ry -25 rz 23.9 deg; joints [-0.828, -48.531, 101.78, 38.397, -108.064, -4.356, -783.901]
  MoveL 271 to (-40.75, 186.98, 170) mm, rotated rx -90 ry -25 rz 17.11 deg; joints [-1.185, -48.702, 102.087, 38.193, -108.039, -4.092, -777.113]
  MoveL 272 to (-48.24, 192.12, 160) mm, rotated rx -90 ry -25 rz 10.19 deg; joints [-1.544, -48.873, 102.387, 37.985, -108.009, -3.831, -770.193]
  MoveL 273 to (-55.2, 198.19, 150) mm, rotated rx -90 ry -25 rz 3.18 deg; joints [-1.904, -49.043, 102.68, 37.775, -107.975, -3.574, -763.183]
  MoveL 274 to (-61.48, 205.13, 140) mm, rotated rx -90 ry -25 rz -3.87 deg; joints [-2.265, -49.212, 102.967, 37.562, -107.937, -3.321, -756.127]
  MoveL 275 to (-66.92, 212.81, 130) mm, rotated rx -90 ry -25 rz -10.94 deg; joints [-2.628, -49.38, 103.247, 37.346, -107.896, -3.07, -749.064]
  MoveL 276 to (-71.41, 221.1, 120) mm, rotated rx -90 ry -25 rz -17.96 deg; joints [-2.992, -49.546, 103.52, 37.128, -107.851, -2.823, -742.035]
  MoveL 277 to (-74.87, 229.83, 110) mm, rotated rx -90 ry -25 rz -24.92 deg; joints [-3.358, -49.71, 103.787, 36.907, -107.804, -2.577, -735.078]
  MoveL 278 to (-77.24, 238.83, 100) mm, rotated rx -90 ry -25 rz -31.77 deg; joints [-3.725, -49.872, 104.048, 36.684, -107.755, -2.334, -728.229]
  MoveL 279 to (-78.53, 247.91, 90) mm, rotated rx -90 ry -25 rz -38.48 deg; joints [-4.093, -50.03, 104.302, 36.459, -107.704, -2.093, -721.522]
  MoveL 280 to (-78.77, 256.9, 80) mm, rotated rx -90 ry -25 rz -45.01 deg; joints [-4.463, -50.185, 104.551, 36.231, -107.651, -1.852, -714.991]
  MoveL 281 to (-78, 265.63, 70) mm, rotated rx -90 ry -25 rz -51.33 deg; joints [-4.834, -50.336, 104.793, 36.002, -107.597, -1.613, -708.666]
  MoveL 282 to (-76.35, 273.96, 60) mm, rotated rx -90 ry -25 rz -57.42 deg; joints [-5.207, -50.483, 105.028, 35.77, -107.542, -1.374, -702.579]
  MoveL 283 to (-73.92, 281.75, 50) mm, rotated rx -90 ry -25 rz -63.24 deg; joints [-5.581, -50.625, 105.258, 35.538, -107.487, -1.136, -696.759]
  MoveL 284 to (-70.87, 288.9, 40) mm, rotated rx -90 ry -25 rz -68.76 deg; joints [-5.956, -50.762, 105.482, 35.303, -107.432, -0.898, -691.235]
  MoveL 285 to (-67.34, 295.36, 30) mm, rotated rx -90 ry -25 rz -73.96 deg; joints [-6.332, -50.894, 105.7, 35.067, -107.377, -0.661, -686.036]
  MoveL 286 to (-63.51, 301.08, 20) mm, rotated rx -90 ry -25 rz -78.81 deg; joints [-6.709, -51.021, 105.911, 34.829, -107.322, -0.423, -681.192]
  MoveL 287 to (-59.54, 306.05, 10) mm, rotated rx -90 ry -25 rz -83.27 deg; joints [-7.088, -51.143, 106.117, 34.59, -107.267, -0.186, -676.73]
  MoveL 288 to (-55.59, 310.29, 0) mm, rotated rx -90 ry -25 rz -87.32 deg; joints [-7.468, -51.259, 106.317, 34.349, -107.213, 0.052, -672.681]
  Set speed (1000.0 mm/s)
  MoveL 289 to (-55.59, 310.29, 0) mm, rotated rx -90 ry -25 rz -87.32 deg; joints [-7.468, -51.259, 106.317, 34.349, -107.213, 0.052, -672.681]
  Set speed (1000.0 mm/s)
  MoveL 290 to (34.79, 183.72, 290) mm, rotated rx -90 ry -25 rz 77.69 deg; joints [2.992, -46.56, 97.967, 40.451, -108.125, -7.483, -837.692]
  MoveL 291 to (34.79, 183.72, 290) mm, rotated rx -90 ry -25 rz 77.69 deg; joints [2.992, -46.56, 97.967, 40.451, -108.125, -7.483, -837.692]
  Set speed (60.0 mm/s)
  MoveL 292 to (30.72, 204.12, 290) mm, rotated rx -90 ry -25 rz 83.8 deg; joints [2.992, -45.676, 98.058, 40.663, -108.866, -6.815, -843.801]
  Set speed (1000.0 mm/s)
  MoveL 293 to (30.72, 204.12, 290) mm, rotated rx -90 ry -25 rz 83.8 deg; joints [2.992, -45.676, 98.058, 40.663, -108.866, -6.815, -843.801]
  Set speed (1000.0 mm/s)
  MoveL 294 to (-55.59, 310.29, 0) mm, rotated rx -90 ry -25 rz -87.32 deg; joints [-7.468, -51.259, 106.317, 34.349, -107.213, 0.052, -672.681]
  MoveL 295 to (-55.59, 310.29, 0) mm, rotated rx -90 ry -25 rz -87.32 deg; joints [-7.468, -51.259, 106.317, 34.349, -107.213, 0.052, -672.681]
  Set speed (60.0 mm/s)
  MoveL 296 to (-45.21, 292.27, 0) mm, rotated rx -90 ry -25 rz -83.07 deg; joints [-7.468, -50.285, 106.421, 34.543, -108.102, 0.692, -676.927]
  Set speed (1000.0 mm/s)
  MoveL 297 to (-45.21, 292.27, 0) mm, rotated rx -90 ry -25 rz -83.07 deg; joints [-7.468, -50.285, 106.421, 34.543, -108.102, 0.692, -676.927]
  Set speed (1000.0 mm/s)
  MoveL 298 to (-55.59, 310.29, 0) mm, rotated rx -90 ry -25 rz -87.32 deg; joints [-7.468, -51.259, 106.317, 34.349, -107.213, 0.052, -672.681]
  MoveL 299 to (-55.59, 310.29, 0) mm, rotated rx -90 ry -25 rz -87.32 deg; joints [-7.468, -51.259, 106.317, 34.349, -107.213, 0.052, -672.681]
  Set speed (60.0 mm/s)
  MoveL 300 to (-59.54, 306.05, 10) mm, rotated rx -90 ry -25 rz -83.27 deg; joints [-7.088, -51.143, 106.117, 34.59, -107.267, -0.186, -676.73]
  MoveL 301 to (-63.51, 301.08, 20) mm, rotated rx -90 ry -25 rz -78.81 deg; joints [-6.709, -51.021, 105.911, 34.829, -107.322, -0.423, -681.192]
  MoveL 302 to (-67.34, 295.36, 30) mm, rotated rx -90 ry -25 rz -73.96 deg; joints [-6.332, -50.894, 105.7, 35.067, -107.377, -0.661, -686.036]
  MoveL 303 to (-70.87, 288.9, 40) mm, rotated rx -90 ry -25 rz -68.76 deg; joints [-5.956, -50.762, 105.482, 35.303, -107.432, -0.898, -691.235]
  MoveL 304 to (-73.92, 281.75, 50) mm, rotated rx -90 ry -25 rz -63.24 deg; joints [-5.581, -50.625, 105.258, 35.538, -107.487, -1.136, -696.759]
  MoveL 305 to (-76.35, 273.96, 60) mm, rotated rx -90 ry -25 rz -57.42 deg; joints [-5.207, -50.483, 105.028, 35.77, -107.542, -1.374, -702.579]
  MoveL 306 to (-78, 265.63, 70) mm, rotated rx -90 ry -25 rz -51.33 deg; joints [-4.834, -50.336, 104.793, 36.002, -107.597, -1.613, -708.666]
  MoveL 307 to (-78.77, 256.9, 80) mm, rotated rx -90 ry -25 rz -45.01 deg; joints [-4.463, -50.185, 104.551, 36.231, -107.651, -1.852, -714.991]
  MoveL 308 to (-78.53, 247.91, 90) mm, rotated rx -90 ry -25 rz -38.48 deg; joints [-4.093, -50.03, 104.302, 36.459, -107.704, -2.093, -721.522]
  MoveL 309 to (-77.24, 238.83, 100) mm, rotated rx -90 ry -25 rz -31.77 deg; joints [-3.725, -49.872, 104.048, 36.684, -107.755, -2.334, -728.229]
  MoveL 310 to (-74.87, 229.83, 110) mm, rotated rx -90 ry -25 rz -24.92 deg; joints [-3.358, -49.71, 103.787, 36.907, -107.804, -2.577, -735.078]
  MoveL 311 to (-71.41, 221.1, 120) mm, rotated rx -90 ry -25 rz -17.96 deg; joints [-2.992, -49.546, 103.52, 37.128, -107.851, -2.823, -742.035]
  MoveL 312 to (-66.92, 212.81, 130) mm, rotated rx -90 ry -25 rz -10.94 deg; joints [-2.628, -49.38, 103.247, 37.346, -107.896, -3.07, -749.064]
  MoveL 313 to (-61.48, 205.13, 140) mm, rotated rx -90 ry -25 rz -3.87 deg; joints [-2.265, -49.212, 102.967, 37.562, -107.937, -3.321, -756.127]
  MoveL 314 to (-55.2, 198.19, 150) mm, rotated rx -90 ry -25 rz 3.18 deg; joints [-1.904, -49.043, 102.68, 37.775, -107.975, -3.574, -763.183]
  MoveL 315 to (-48.24, 192.12, 160) mm, rotated rx -90 ry -25 rz 10.19 deg; joints [-1.544, -48.873, 102.387, 37.985, -108.009, -3.831, -770.193]
  MoveL 316 to (-40.75, 186.98, 170) mm, rotated rx -90 ry -25 rz 17.11 deg; joints [-1.185, -48.702, 102.087, 38.193, -108.039, -4.092, -777.113]
  MoveL 317 to (-32.91, 182.83, 180) mm, rotated rx -90 ry -25 rz 23.9 deg; joints [-0.828, -48.531, 101.78, 38.397, -108.064, -4.356, -783.901]
  MoveL 318 to (-24.89, 179.66, 190) mm, rotated rx -90 ry -25 rz 30.51 deg; joints [-0.473, -48.36, 101.467, 38.598, -108.086, -4.624, -790.512]
  MoveL 319 to (-16.88, 177.46, 200) mm, rotated rx -90 ry -25 rz 36.9 deg; joints [-0.119, -48.187, 101.147, 38.797, -108.104, -4.896, -796.902]
  MoveL 320 to (-9.03, 176.15, 210) mm, rotated rx -90 ry -25 rz 43.03 deg; joints [0.233, -48.014, 100.82, 38.992, -108.118, -5.172, -803.03]
  MoveL 321 to (-1.49, 175.64, 220) mm, rotated rx -90 ry -25 rz 48.85 deg; joints [0.584, -47.84, 100.487, 39.184, -108.128, -5.451, -808.851]
  MoveL 322 to (5.61, 175.83, 230) mm, rotated rx -90 ry -25 rz 54.33 deg; joints [0.933, -47.665, 100.147, 39.373, -108.135, -5.733, -814.325]
  MoveL 323 to (12.17, 176.57, 240) mm, rotated rx -90 ry -25 rz 59.41 deg; joints [1.28, -47.487, 99.8, 39.56, -108.139, -6.019, -819.412]
  MoveL 324 to (18.11, 177.74, 250) mm, rotated rx -90 ry -25 rz 64.07 deg; joints [1.626, -47.308, 99.447, 39.743, -108.14, -6.307, -824.071]
  MoveL 325 to (23.38, 179.17, 260) mm, rotated rx -90 ry -25 rz 68.27 deg; joints [1.97, -47.126, 99.087, 39.924, -108.139, -6.598, -828.265]
  MoveL 326 to (27.92, 180.74, 270) mm, rotated rx -90 ry -25 rz 71.96 deg; joints [2.312, -46.941, 98.72, 40.102, -108.136, -6.891, -831.958]
  MoveL 327 to (31.73, 182.3, 280) mm, rotated rx -90 ry -25 rz 75.11 deg; joints [2.653, -46.752, 98.347, 40.278, -108.131, -7.186, -835.112]
  MoveL 328 to (34.79, 183.72, 290) mm, rotated rx -90 ry -25 rz 77.69 deg; joints [2.992, -46.56, 97.967, 40.451, -108.125, -7.483, -837.692]
  Set speed (1000.0 mm/s)
  MoveL 329 to (34.79, 183.72, 290) mm, rotated rx -90 ry -25 rz 77.69 deg; joints [2.992, -46.56, 97.967, 40.451, -108.125, -7.483, -837.692]
  Set speed (1000.0 mm/s)
  MoveL 330 to (30.72, 204.12, 290) mm, rotated rx -90 ry -25 rz 83.8 deg; joints [2.992, -45.676, 98.058, 40.663, -108.866, -6.815, -843.801]
  MoveL 331 to (30.72, 204.12, 290) mm, rotated rx -90 ry -25 rz 83.8 deg; joints [2.992, -45.676, 98.058, 40.663, -108.866, -6.815, -843.801]
  Set speed (60.0 mm/s)
  MoveL 332 to (28.54, 202.85, 280) mm, rotated rx -90 ry -25 rz 81.18 deg; joints [2.653, -45.864, 98.438, 40.49, -108.877, -6.518, -841.184]
  MoveL 333 to (25.81, 201.43, 270) mm, rotated rx -90 ry -25 rz 77.98 deg; joints [2.312, -46.049, 98.811, 40.314, -108.886, -6.222, -837.983]
  MoveL 334 to (22.53, 199.96, 260) mm, rotated rx -90 ry -25 rz 74.23 deg; joints [1.97, -46.229, 99.177, 40.136, -108.895, -5.929, -834.232]
  MoveL 335 to (18.7, 198.53, 250) mm, rotated rx -90 ry -25 rz 69.97 deg; joints [1.626, -46.407, 99.537, 39.956, -108.901, -5.637, -829.967]
  MoveL 336 to (14.35, 197.26, 240) mm, rotated rx -90 ry -25 rz 65.22 deg; joints [1.28, -46.582, 99.89, 39.772, -108.905, -5.349, -825.225]
  MoveL 337 to (9.52, 196.26, 230) mm, rotated rx -90 ry -25 rz 60.04 deg; joints [0.933, -46.755, 100.237, 39.586, -108.907, -5.063, -820.042]
  MoveL 338 to (4.24, 195.64, 220) mm, rotated rx -90 ry -25 rz 54.46 deg; joints [0.584, -46.926, 100.577, 39.397, -108.906, -4.78, -814.46]
  MoveL 339 to (-1.41, 195.5, 210) mm, rotated rx -90 ry -25 rz 48.52 deg; joints [0.233, -47.095, 100.911, 39.205, -108.901, -4.5, -808.518]
  MoveL 340 to (-7.35, 195.94, 200) mm, rotated rx -90 ry -25 rz 42.26 deg; joints [-0.119, -47.264, 101.238, 39.01, -108.893, -4.224, -802.261]
  MoveL 341 to (-13.47, 197.04, 190) mm, rotated rx -90 ry -25 rz 35.73 deg; joints [-0.473, -47.431, 101.558, 38.812, -108.882, -3.952, -795.734]
  MoveL 342 to (-19.65, 198.85, 180) mm, rotated rx -90 ry -25 rz 28.98 deg; joints [-0.828, -47.598, 101.872, 38.61, -108.866, -3.684, -788.982]
  MoveL 343 to (-25.78, 201.42, 170) mm, rotated rx -90 ry -25 rz 22.05 deg; joints [-1.185, -47.765, 102.179, 38.406, -108.847, -3.419, -782.053]
  MoveL 344 to (-31.7, 204.73, 160) mm, rotated rx -90 ry -25 rz 14.99 deg; joints [-1.544, -47.932, 102.48, 38.198, -108.823, -3.159, -774.993]
  MoveL 345 to (-37.3, 208.79, 150) mm, rotated rx -90 ry -25 rz 7.85 deg; joints [-1.904, -48.098, 102.774, 37.987, -108.795, -2.902, -767.85]
  MoveL 346 to (-42.45, 213.53, 140) mm, rotated rx -90 ry -25 rz 0.67 deg; joints [-2.265, -48.263, 103.061, 37.774, -108.763, -2.649, -760.67]
  MoveL 347 to (-47.02, 218.88, 130) mm, rotated rx -90 ry -25 rz -6.5 deg; joints [-2.628, -48.428, 103.342, 37.557, -108.727, -2.399, -753.496]
  MoveL 348 to (-50.93, 224.75, 120) mm, rotated rx -90 ry -25 rz -13.63 deg; joints [-2.992, -48.591, 103.616, 37.338, -108.689, -2.153, -746.37]
  MoveL 349 to (-54.1, 231.02, 110) mm, rotated rx -90 ry -25 rz -20.67 deg; joints [-3.358, -48.752, 103.884, 37.116, -108.647, -1.909, -739.332]
  MoveL 350 to (-56.49, 237.56, 100) mm, rotated rx -90 ry -25 rz -27.58 deg; joints [-3.725, -48.911, 104.146, 36.892, -108.602, -1.667, -732.418]
  MoveL 351 to (-58.06, 244.24, 90) mm, rotated rx -90 ry -25 rz -34.34 deg; joints [-4.093, -49.068, 104.401, 36.666, -108.556, -1.427, -725.663]
  MoveL 352 to (-58.85, 250.92, 80) mm, rotated rx -90 ry -25 rz -40.9 deg; joints [-4.463, -49.221, 104.65, 36.437, -108.508, -1.189, -719.1]
  MoveL 353 to (-58.87, 257.48, 70) mm, rotated rx -90 ry -25 rz -47.24 deg; joints [-4.834, -49.37, 104.893, 36.206, -108.459, -0.952, -712.759]
  MoveL 354 to (-58.2, 263.79, 60) mm, rotated rx -90 ry -25 rz -53.33 deg; joints [-5.207, -49.515, 105.13, 35.974, -108.409, -0.716, -706.668]
  MoveL 355 to (-56.92, 269.76, 50) mm, rotated rx -90 ry -25 rz -59.14 deg; joints [-5.581, -49.656, 105.36, 35.739, -108.358, -0.48, -700.857]
  MoveL 356 to (-55.13, 275.3, 40) mm, rotated rx -90 ry -25 rz -64.65 deg; joints [-5.956, -49.792, 105.585, 35.503, -108.307, -0.245, -695.351]
  MoveL 357 to (-52.95, 280.35, 30) mm, rotated rx -90 ry -25 rz -69.82 deg; joints [-6.332, -49.923, 105.803, 35.266, -108.256, -0.01, -690.178]
  MoveL 358 to (-50.48, 284.87, 20) mm, rotated rx -90 ry -25 rz -74.63 deg; joints [-6.709, -50.049, 106.015, 35.026, -108.204, 0.224, -685.365]
  MoveL 359 to (-47.86, 288.84, 10) mm, rotated rx -90 ry -25 rz -79.06 deg; joints [-7.088, -50.169, 106.221, 34.785, -108.153, 0.458, -680.939]
  MoveL 360 to (-45.21, 292.27, 0) mm, rotated rx -90 ry -25 rz -83.07 deg; joints [-7.468, -50.285, 106.421, 34.543, -108.102, 0.692, -676.927]
  Set speed (1000.0 mm/s)
  MoveL 361 to (-45.21, 292.27, 0) mm, rotated rx -90 ry -25 rz -83.07 deg; joints [-7.468, -50.285, 106.421, 34.543, -108.102, 0.692, -676.927]
  Set speed (1000.0 mm/s)
  MoveL 362 to (30.72, 204.12, 290) mm, rotated rx -90 ry -25 rz 83.8 deg; joints [2.992, -45.676, 98.058, 40.663, -108.866, -6.815, -843.801]
  MoveL 363 to (30.72, 204.12, 290) mm, rotated rx -90 ry -25 rz 83.8 deg; joints [2.992, -45.676, 98.058, 40.663, -108.866, -6.815, -843.801]
  Set speed (60.0 mm/s)
  MoveL 364 to (58.22, 245.2, 290) mm, rotated rx -90 ry -25 rz 135.28 deg; joints [2.992, -45.821, 98.045, 40.627, -108.746, -6.924, -895.284]
  Set speed (1000.0 mm/s)
  MoveL 365 to (58.22, 245.2, 290) mm, rotated rx -90 ry -25 rz 135.28 deg; joints [2.992, -45.821, 98.045, 40.627, -108.746, -6.924, -895.284]
  Set speed (1000.0 mm/s)
  MoveL 366 to (-45.21, 292.27, 0) mm, rotated rx -90 ry -25 rz -83.07 deg; joints [-7.468, -50.285, 106.421, 34.543, -108.102, 0.692, -1036.927]
  MoveL 367 to (-45.21, 292.27, 0) mm, rotated rx -90 ry -25 rz -83.07 deg; joints [-7.468, -50.285, 106.421, 34.543, -108.102, 0.692, -1036.927]
  Set speed (60.0 mm/s)
  MoveL 368 to (-58.12, 244.54, 0) mm, rotated rx -90 ry -25 rz -34.64 deg; joints [-7.468, -50.113, 106.436, 34.578, -108.256, 0.804, -1085.364]
  Set speed (1000.0 mm/s)
  MoveL 369 to (-58.12, 244.54, 0) mm, rotated rx -90 ry -25 rz -34.64 deg; joints [-7.468, -50.113, 106.436, 34.578, -108.256, 0.804, -1085.364]
  Set speed (1000.0 mm/s)
  MoveL 370 to (-45.21, 292.27, 0) mm, rotated rx -90 ry -25 rz -83.07 deg; joints [-7.468, -50.285, 106.421, 34.543, -108.102, 0.692, -1036.927]
  MoveL 371 to (-45.21, 292.27, 0) mm, rotated rx -90 ry -25 rz -83.07 deg; joints [-7.468, -50.285, 106.421, 34.543, -108.102, 0.692, -1036.927]
  Set speed (60.0 mm/s)
  MoveL 372 to (-47.86, 288.84, 10) mm, rotated rx -90 ry -25 rz -79.06 deg; joints [-7.088, -50.169, 106.221, 34.785, -108.153, 0.458, -1040.939]
  MoveL 373 to (-50.48, 284.87, 20) mm, rotated rx -90 ry -25 rz -74.63 deg; joints [-6.709, -50.049, 106.015, 35.026, -108.204, 0.224, -1045.365]
  MoveL 374 to (-52.95, 280.35, 30) mm, rotated rx -90 ry -25 rz -69.82 deg; joints [-6.332, -49.923, 105.803, 35.266, -108.256, -0.01, -1050.178]
  MoveL 375 to (-55.13, 275.3, 40) mm, rotated rx -90 ry -25 rz -64.65 deg; joints [-5.956, -49.792, 105.585, 35.503, -108.307, -0.245, -1055.351]
  MoveL 376 to (-56.92, 269.76, 50) mm, rotated rx -90 ry -25 rz -59.14 deg; joints [-5.581, -49.656, 105.36, 35.739, -108.358, -0.48, -1060.857]
  MoveL 377 to (-58.2, 263.79, 60) mm, rotated rx -90 ry -25 rz -53.33 deg; joints [-5.207, -49.515, 105.13, 35.974, -108.409, -0.716, -1066.668]
  MoveL 378 to (-58.87, 257.48, 70) mm, rotated rx -90 ry -25 rz -47.24 deg; joints [-4.834, -49.37, 104.893, 36.206, -108.459, -0.952, -1072.759]
  MoveL 379 to (-58.85, 250.92, 80) mm, rotated rx -90 ry -25 rz -40.9 deg; joints [-4.463, -49.221, 104.65, 36.437, -108.508, -1.189, -1079.1]
  MoveL 380 to (-58.06, 244.24, 90) mm, rotated rx -90 ry -25 rz -34.34 deg; joints [-4.093, -49.068, 104.401, 36.666, -108.556, -1.427, -1085.663]
  MoveL 381 to (-56.49, 237.56, 100) mm, rotated rx -90 ry -25 rz -27.58 deg; joints [-3.725, -48.911, 104.146, 36.892, -108.602, -1.667, -1092.418]
  MoveL 382 to (-54.1, 231.02, 110) mm, rotated rx -90 ry -25 rz -20.67 deg; joints [-3.358, -48.752, 103.884, 37.116, -108.647, -1.909, -1099.332]
  MoveL 383 to (-50.93, 224.75, 120) mm, rotated rx -90 ry -25 rz -13.63 deg; joints [-2.992, -48.591, 103.616, 37.338, -108.689, -2.153, -1106.37]
  MoveL 384 to (-47.02, 218.88, 130) mm, rotated rx -90 ry -25 rz -6.5 deg; joints [-2.628, -48.428, 103.342, 37.557, -108.727, -2.399, -1113.496]
  MoveL 385 to (-42.45, 213.53, 140) mm, rotated rx -90 ry -25 rz 0.67 deg; joints [-2.265, -48.263, 103.061, 37.774, -108.763, -2.649, -1120.67]
  MoveL 386 to (-37.3, 208.79, 150) mm, rotated rx -90 ry -25 rz 7.85 deg; joints [-1.904, -48.098, 102.774, 37.987, -108.795, -2.902, -1127.85]
  MoveL 387 to (-31.7, 204.73, 160) mm, rotated rx -90 ry -25 rz 14.99 deg; joints [-1.544, -47.932, 102.48, 38.198, -108.823, -3.159, -1134.993]
  MoveL 388 to (-25.78, 201.42, 170) mm, rotated rx -90 ry -25 rz 22.05 deg; joints [-1.185, -47.765, 102.179, 38.406, -108.847, -3.419, -1142.053]
  MoveL 389 to (-19.65, 198.85, 180) mm, rotated rx -90 ry -25 rz 28.98 deg; joints [-0.828, -47.598, 101.872, 38.61, -108.866, -3.684, -1148.982]
  MoveL 390 to (-13.47, 197.04, 190) mm, rotated rx -90 ry -25 rz 35.73 deg; joints [-0.473, -47.431, 101.558, 38.812, -108.882, -3.952, -1155.734]
  MoveL 391 to (-7.35, 195.94, 200) mm, rotated rx -90 ry -25 rz 42.26 deg; joints [-0.119, -47.264, 101.238, 39.01, -108.893, -4.224, -1162.261]
  MoveL 392 to (-1.41, 195.5, 210) mm, rotated rx -90 ry -25 rz 48.52 deg; joints [0.233, -47.095, 100.911, 39.205, -108.901, -4.5, -1168.518]
  MoveL 393 to (4.24, 195.64, 220) mm, rotated rx -90 ry -25 rz 54.46 deg; joints [0.584, -46.926, 100.577, 39.397, -108.906, -4.78, -1174.46]
  MoveL 394 to (9.52, 196.26, 230) mm, rotated rx -90 ry -25 rz 60.04 deg; joints [0.933, -46.755, 100.237, 39.586, -108.907, -5.063, -1180.042]
  MoveL 395 to (14.35, 197.26, 240) mm, rotated rx -90 ry -25 rz 65.22 deg; joints [1.28, -46.582, 99.89, 39.772, -108.905, -5.349, -1185.225]
  MoveL 396 to (18.7, 198.53, 250) mm, rotated rx -90 ry -25 rz 69.97 deg; joints [1.626, -46.407, 99.537, 39.956, -108.901, -5.637, -1189.967]
  MoveL 397 to (22.53, 199.96, 260) mm, rotated rx -90 ry -25 rz 74.23 deg; joints [1.97, -46.229, 99.177, 40.136, -108.895, -5.929, -1194.232]
  MoveL 398 to (25.81, 201.43, 270) mm, rotated rx -90 ry -25 rz 77.98 deg; joints [2.312, -46.049, 98.811, 40.314, -108.886, -6.222, -1197.983]
  MoveL 399 to (28.54, 202.85, 280) mm, rotated rx -90 ry -25 rz 81.18 deg; joints [2.653, -45.864, 98.438, 40.49, -108.877, -6.518, -1201.184]
  MoveL 400 to (30.72, 204.12, 290) mm, rotated rx -90 ry -25 rz 83.8 deg; joints [2.992, -45.676, 98.058, 40.663, -108.866, -6.815, -1203.801]
  Set speed (1000.0 mm/s)
  MoveL 401 to (30.72, 204.12, 290) mm, rotated rx -90 ry -25 rz 83.8 deg; joints [2.992, -45.676, 98.058, 40.663, -108.866, -6.815, -1203.801]
  Set speed (1000.0 mm/s)
  MoveL 402 to (58.22, 245.2, 290) mm, rotated rx -90 ry -25 rz 135.28 deg; joints [2.992, -45.821, 98.045, 40.627, -108.746, -6.924, -1255.284]
  MoveL 403 to (58.22, 245.2, 290) mm, rotated rx -90 ry -25 rz 135.28 deg; joints [2.992, -45.821, 98.045, 40.627, -108.746, -6.924, -1255.284]
  Set speed (60.0 mm/s)
  MoveL 404 to (57.77, 242.72, 280) mm, rotated rx -90 ry -25 rz 132.81 deg; joints [2.653, -46.006, 98.425, 40.456, -108.759, -6.624, -1252.814]
  MoveL 405 to (57.08, 239.72, 270) mm, rotated rx -90 ry -25 rz 129.79 deg; joints [2.312, -46.186, 98.799, 40.282, -108.773, -6.324, -1249.788]
  MoveL 406 to (56.08, 236.26, 260) mm, rotated rx -90 ry -25 rz 126.23 deg; joints [1.97, -46.361, 99.166, 40.105, -108.786, -6.025, -1246.235]
  MoveL 407 to (54.69, 232.42, 250) mm, rotated rx -90 ry -25 rz 122.18 deg; joints [1.626, -46.53, 99.527, 39.927, -108.798, -5.728, -1242.184]
  MoveL 408 to (52.84, 228.29, 240) mm, rotated rx -90 ry -25 rz 117.66 deg; joints [1.28, -46.696, 99.881, 39.746, -108.81, -5.432, -1237.664]
  MoveL 409 to (50.46, 223.96, 230) mm, rotated rx -90 ry -25 rz 112.71 deg; joints [0.933, -46.857, 100.229, 39.562, -108.822, -5.137, -1232.705]
  MoveL 410 to (47.51, 219.54, 220) mm, rotated rx -90 ry -25 rz 107.34 deg; joints [0.584, -47.015, 100.57, 39.376, -108.831, -4.844, -1227.337]
  MoveL 411 to (43.95, 215.15, 210) mm, rotated rx -90 ry -25 rz 101.59 deg; joints [0.233, -47.169, 100.905, 39.188, -108.84, -4.553, -1221.59]
  MoveL 412 to (39.77, 210.92, 200) mm, rotated rx -90 ry -25 rz 95.5 deg; joints [-0.119, -47.32, 101.233, 38.997, -108.846, -4.265, -1215.499]
  MoveL 413 to (34.96, 206.97, 190) mm, rotated rx -90 ry -25 rz 89.1 deg; joints [-0.473, -47.469, 101.555, 38.803, -108.85, -3.979, -1209.096]
  MoveL 414 to (29.57, 203.44, 180) mm, rotated rx -90 ry -25 rz 82.42 deg; joints [-0.828, -47.616, 101.871, 38.606, -108.852, -3.696, -1202.421]
  MoveL 415 to (23.65, 200.44, 170) mm, rotated rx -90 ry -25 rz 75.51 deg; joints [-1.185, -47.761, 102.18, 38.406, -108.85, -3.417, -1195.511]
  MoveL 416 to (17.28, 198.07, 160) mm, rotated rx -90 ry -25 rz 68.41 deg; joints [-1.544, -47.906, 102.482, 38.204, -108.844, -3.141, -1188.409]
  MoveL 417 to (10.57, 196.44, 150) mm, rotated rx -90 ry -25 rz 61.16 deg; joints [-1.904, -48.051, 102.777, 37.998, -108.835, -2.869, -1181.159]
  MoveL 418 to (3.62, 195.59, 140) mm, rotated rx -90 ry -25 rz 53.81 deg; joints [-2.265, -48.195, 103.067, 37.789, -108.821, -2.601, -1173.808]
  MoveL 419 to (-3.42, 195.58, 130) mm, rotated rx -90 ry -25 rz 46.4 deg; joints [-2.628, -48.339, 103.349, 37.577, -108.803, -2.338, -1166.404]
  MoveL 420 to (-10.42, 196.41, 120) mm, rotated rx -90 ry -25 rz 38.99 deg; joints [-2.992, -48.483, 103.625, 37.362, -108.781, -2.078, -1158.993]
  MoveL 421 to (-17.25, 198.06, 110) mm, rotated rx -90 ry -25 rz 31.62 deg; joints [-3.358, -48.627, 103.895, 37.144, -108.754, -1.823, -1151.625]
  MoveL 422 to (-23.78, 200.49, 100) mm, rotated rx -90 ry -25 rz 24.35 deg; joints [-3.725, -48.771, 104.157, 36.923, -108.724, -1.571, -1144.346]
  MoveL 423 to (-29.89, 203.62, 90) mm, rotated rx -90 ry -25 rz 17.2 deg; joints [-4.093, -48.915, 104.414, 36.699, -108.689, -1.323, -1137.203]
  MoveL 424 to (-35.48, 207.36, 80) mm, rotated rx -90 ry -25 rz 10.24 deg; joints [-4.463, -49.058, 104.664, 36.472, -108.65, -1.078, -1130.238]
  MoveL 425 to (-40.49, 211.59, 70) mm, rotated rx -90 ry -25 rz 3.49 deg; joints [-4.834, -49.199, 104.907, 36.243, -108.608, -0.837, -1123.492]
  MoveL 426 to (-44.86, 216.19, 60) mm, rotated rx -90 ry -25 rz -3 deg; joints [-5.207, -49.339, 105.145, 36.011, -108.563, -0.597, -1117.004]
  MoveL 427 to (-48.58, 221.03, 50) mm, rotated rx -90 ry -25 rz -9.19 deg; joints [-5.581, -49.477, 105.375, 35.777, -108.516, -0.36, -1110.81]
  MoveL 428 to (-51.63, 225.99, 40) mm, rotated rx -90 ry -25 rz -15.06 deg; joints [-5.956, -49.611, 105.6, 35.541, -108.466, -0.125, -1104.943]
  MoveL 429 to (-54.06, 230.92, 30) mm, rotated rx -90 ry -25 rz -20.56 deg; joints [-6.332, -49.743, 105.818, 35.303, -108.415, 0.109, -1099.435]
  MoveL 430 to (-55.91, 235.73, 20) mm, rotated rx -90 ry -25 rz -25.68 deg; joints [-6.709, -49.87, 106.03, 35.063, -108.363, 0.341, -1094.317]
  MoveL 431 to (-57.23, 240.3, 10) mm, rotated rx -90 ry -25 rz -30.38 deg; joints [-7.088, -49.994, 106.236, 34.821, -108.31, 0.573, -1089.617]
  MoveL 432 to (-58.12, 244.54, 0) mm, rotated rx -90 ry -25 rz -34.64 deg; joints [-7.468, -50.113, 106.436, 34.578, -108.256, 0.804, -1085.364]
  Set speed (1000.0 mm/s)
  MoveL 433 to (-58.12, 244.54, 0) mm, rotated rx -90 ry -25 rz -34.64 deg; joints [-7.468, -50.113, 106.436, 34.578, -108.256, 0.804, -1085.364]
  Set speed (1000.0 mm/s)
  MoveL 434 to (58.22, 245.2, 290) mm, rotated rx -90 ry -25 rz 135.28 deg; joints [2.992, -45.821, 98.045, 40.627, -108.746, -6.924, -1255.284]
  MoveL 435 to (58.22, 245.2, 290) mm, rotated rx -90 ry -25 rz 135.28 deg; joints [2.992, -45.821, 98.045, 40.627, -108.746, -6.924, -1255.284]
  Set speed (60.0 mm/s)
  MoveL 436 to (78.63, 249.2, 290) mm, rotated rx -90 ry -25 rz 139.42 deg; joints [2.992, -46.728, 97.946, 40.411, -107.981, -7.612, -1259.419]
  Set speed (1000.0 mm/s)
  MoveL 437 to (78.63, 249.2, 290) mm, rotated rx -90 ry -25 rz 139.42 deg; joints [2.992, -46.728, 97.946, 40.411, -107.981, -7.612, -1259.419]
  Set speed (1000.0 mm/s)
  MoveL 438 to (-58.12, 244.54, 0) mm, rotated rx -90 ry -25 rz -34.64 deg; joints [-7.468, -50.113, 106.436, 34.578, -108.256, 0.804, -1085.364]
  MoveL 439 to (-58.12, 244.54, 0) mm, rotated rx -90 ry -25 rz -34.64 deg; joints [-7.468, -50.113, 106.436, 34.578, -108.256, 0.804, -1085.364]
  Set speed (60.0 mm/s)
  MoveL 440 to (-76.17, 234.21, 0) mm, rotated rx -90 ry -25 rz -28.29 deg; joints [-7.468, -51.057, 106.341, 34.389, -107.4, 0.186, -1091.709]
  Set speed (1000.0 mm/s)
  MoveL 441 to (-76.17, 234.21, 0) mm, rotated rx -90 ry -25 rz -28.29 deg; joints [-7.468, -51.057, 106.341, 34.389, -107.4, 0.186, -1091.709]
  Set speed (1000.0 mm/s)
  MoveL 442 to (-58.12, 244.54, 0) mm, rotated rx -90 ry -25 rz -34.64 deg; joints [-7.468, -50.113, 106.436, 34.578, -108.256, 0.804, -1085.364]
  MoveL 443 to (-58.12, 244.54, 0) mm, rotated rx -90 ry -25 rz -34.64 deg; joints [-7.468, -50.113, 106.436, 34.578, -108.256, 0.804, -1085.364]
  Set speed (60.0 mm/s)
  MoveL 444 to (-57.23, 240.3, 10) mm, rotated rx -90 ry -25 rz -30.38 deg; joints [-7.088, -49.994, 106.236, 34.821, -108.31, 0.573, -1089.617]
  MoveL 445 to (-55.91, 235.73, 20) mm, rotated rx -90 ry -25 rz -25.68 deg; joints [-6.709, -49.87, 106.03, 35.063, -108.363, 0.341, -1094.317]
  MoveL 446 to (-54.06, 230.92, 30) mm, rotated rx -90 ry -25 rz -20.56 deg; joints [-6.332, -49.743, 105.818, 35.303, -108.415, 0.109, -1099.435]
  MoveL 447 to (-51.63, 225.99, 40) mm, rotated rx -90 ry -25 rz -15.06 deg; joints [-5.956, -49.611, 105.6, 35.541, -108.466, -0.125, -1104.943]
  MoveL 448 to (-48.58, 221.03, 50) mm, rotated rx -90 ry -25 rz -9.19 deg; joints [-5.581, -49.477, 105.375, 35.777, -108.516, -0.36, -1110.81]
  MoveL 449 to (-44.86, 216.19, 60) mm, rotated rx -90 ry -25 rz -3 deg; joints [-5.207, -49.339, 105.145, 36.011, -108.563, -0.597, -1117.004]
  MoveL 450 to (-40.49, 211.59, 70) mm, rotated rx -90 ry -25 rz 3.49 deg; joints [-4.834, -49.199, 104.907, 36.243, -108.608, -0.837, -1123.492]
  MoveL 451 to (-35.48, 207.36, 80) mm, rotated rx -90 ry -25 rz 10.24 deg; joints [-4.463, -49.058, 104.664, 36.472, -108.65, -1.078, -1130.238]
  MoveL 452 to (-29.89, 203.62, 90) mm, rotated rx -90 ry -25 rz 17.2 deg; joints [-4.093, -48.915, 104.414, 36.699, -108.689, -1.323, -1137.203]
  MoveL 453 to (-23.78, 200.49, 100) mm, rotated rx -90 ry -25 rz 24.35 deg; joints [-3.725, -48.771, 104.157, 36.923, -108.724, -1.571, -1144.346]
  MoveL 454 to (-17.25, 198.06, 110) mm, rotated rx -90 ry -25 rz 31.62 deg; joints [-3.358, -48.627, 103.895, 37.144, -108.754, -1.823, -1151.625]
  MoveL 455 to (-10.42, 196.41, 120) mm, rotated rx -90 ry -25 rz 38.99 deg; joints [-2.992, -48.483, 103.625, 37.362, -108.781, -2.078, -1158.993]
  MoveL 456 to (-3.42, 195.58, 130) mm, rotated rx -90 ry -25 rz 46.4 deg; joints [-2.628, -48.339, 103.349, 37.577, -108.803, -2.338, -1166.404]
  MoveL 457 to (3.62, 195.59, 140) mm, rotated rx -90 ry -25 rz 53.81 deg; joints [-2.265, -48.195, 103.067, 37.789, -108.821, -2.601, -1173.808]
  MoveL 458 to (10.57, 196.44, 150) mm, rotated rx -90 ry -25 rz 61.16 deg; joints [-1.904, -48.051, 102.777, 37.998, -108.835, -2.869, -1181.159]
  MoveL 459 to (17.28, 198.07, 160) mm, rotated rx -90 ry -25 rz 68.41 deg; joints [-1.544, -47.906, 102.482, 38.204, -108.844, -3.141, -1188.409]
  MoveL 460 to (23.65, 200.44, 170) mm, rotated rx -90 ry -25 rz 75.51 deg; joints [-1.185, -47.761, 102.18, 38.406, -108.85, -3.417, -1195.511]
  MoveL 461 to (29.57, 203.44, 180) mm, rotated rx -90 ry -25 rz 82.42 deg; joints [-0.828, -47.616, 101.871, 38.606, -108.852, -3.696, -1202.421]
  MoveL 462 to (34.96, 206.97, 190) mm, rotated rx -90 ry -25 rz 89.1 deg; joints [-0.473, -47.469, 101.555, 38.803, -108.85, -3.979, -1209.096]
  MoveL 463 to (39.77, 210.92, 200) mm, rotated rx -90 ry -25 rz 95.5 deg; joints [-0.119, -47.32, 101.233, 38.997, -108.846, -4.265, -1215.499]
  MoveL 464 to (43.95, 215.15, 210) mm, rotated rx -90 ry -25 rz 101.59 deg; joints [0.233, -47.169, 100.905, 39.188, -108.84, -4.553, -1221.59]
  MoveL 465 to (47.51, 219.54, 220) mm, rotated rx -90 ry -25 rz 107.34 deg; joints [0.584, -47.015, 100.57, 39.376, -108.831, -4.844, -1227.337]
  MoveL 466 to (50.46, 223.96, 230) mm, rotated rx -90 ry -25 rz 112.71 deg; joints [0.933, -46.857, 100.229, 39.562, -108.822, -5.137, -1232.705]
  MoveL 467 to (52.84, 228.29, 240) mm, rotated rx -90 ry -25 rz 117.66 deg; joints [1.28, -46.696, 99.881, 39.746, -108.81, -5.432, -1237.664]
  MoveL 468 to (54.69, 232.42, 250) mm, rotated rx -90 ry -25 rz 122.18 deg; joints [1.626, -46.53, 99.527, 39.927, -108.798, -5.728, -1242.184]
  MoveL 469 to (56.08, 236.26, 260) mm, rotated rx -90 ry -25 rz 126.23 deg; joints [1.97, -46.361, 99.166, 40.105, -108.786, -6.025, -1246.235]
  MoveL 470 to (57.08, 239.72, 270) mm, rotated rx -90 ry -25 rz 129.79 deg; joints [2.312, -46.186, 98.799, 40.282, -108.773, -6.324, -1249.788]
  MoveL 471 to (57.77, 242.72, 280) mm, rotated rx -90 ry -25 rz 132.81 deg; joints [2.653, -46.006, 98.425, 40.456, -108.759, -6.624, -1252.814]
  MoveL 472 to (58.22, 245.2, 290) mm, rotated rx -90 ry -25 rz 135.28 deg; joints [2.992, -45.821, 98.045, 40.627, -108.746, -6.924, -1255.284]
  Set speed (1000.0 mm/s)
  MoveL 473 to (58.22, 245.2, 290) mm, rotated rx -90 ry -25 rz 135.28 deg; joints [2.992, -45.821, 98.045, 40.627, -108.746, -6.924, -1255.284]
  Set speed (1000.0 mm/s)
  MoveL 474 to (78.63, 249.2, 290) mm, rotated rx -90 ry -25 rz 139.42 deg; joints [2.992, -46.728, 97.946, 40.411, -107.981, -7.612, -1259.419]
  MoveL 475 to (78.63, 249.2, 290) mm, rotated rx -90 ry -25 rz 139.42 deg; joints [2.992, -46.728, 97.946, 40.411, -107.981, -7.612, -1259.419]
  Set speed (60.0 mm/s)
  MoveL 476 to (78.34, 245.85, 280) mm, rotated rx -90 ry -25 rz 136.96 deg; joints [2.653, -46.916, 98.327, 40.239, -107.991, -7.312, -1256.964]
  MoveL 477 to (77.78, 241.77, 270) mm, rotated rx -90 ry -25 rz 133.96 deg; joints [2.312, -47.099, 98.701, 40.065, -108, -7.012, -1253.959]
  MoveL 478 to (76.86, 237.05, 260) mm, rotated rx -90 ry -25 rz 130.43 deg; joints [1.97, -47.277, 99.068, 39.888, -108.009, -6.712, -1250.435]
  MoveL 479 to (75.48, 231.77, 250) mm, rotated rx -90 ry -25 rz 126.42 deg; joints [1.626, -47.45, 99.43, 39.71, -108.018, -6.414, -1246.422]
  MoveL 480 to (73.51, 226.04, 240) mm, rotated rx -90 ry -25 rz 121.95 deg; joints [1.28, -47.618, 99.784, 39.529, -108.026, -6.117, -1241.95]
  MoveL 481 to (70.88, 219.99, 230) mm, rotated rx -90 ry -25 rz 117.05 deg; joints [0.933, -47.782, 100.133, 39.346, -108.033, -5.821, -1237.052]
  MoveL 482 to (67.49, 213.75, 220) mm, rotated rx -90 ry -25 rz 111.76 deg; joints [0.584, -47.942, 100.475, 39.16, -108.039, -5.526, -1231.756]
  MoveL 483 to (63.28, 207.47, 210) mm, rotated rx -90 ry -25 rz 106.1 deg; joints [0.233, -48.099, 100.81, 38.972, -108.044, -5.234, -1226.097]
  MoveL 484 to (58.22, 201.33, 200) mm, rotated rx -90 ry -25 rz 100.11 deg; joints [-0.119, -48.252, 101.139, 38.782, -108.048, -4.944, -1220.107]
  MoveL 485 to (52.31, 195.49, 190) mm, rotated rx -90 ry -25 rz 93.82 deg; joints [-0.473, -48.403, 101.462, 38.589, -108.049, -4.656, -1213.819]
  MoveL 486 to (45.56, 190.13, 180) mm, rotated rx -90 ry -25 rz 87.27 deg; joints [-0.828, -48.551, 101.778, 38.393, -108.047, -4.371, -1207.271]
  MoveL 487 to (38.04, 185.42, 170) mm, rotated rx -90 ry -25 rz 80.5 deg; joints [-1.185, -48.698, 102.087, 38.194, -108.042, -4.089, -1200.5]
  MoveL 488 to (29.85, 181.5, 160) mm, rotated rx -90 ry -25 rz 73.54 deg; joints [-1.544, -48.844, 102.39, 37.992, -108.034, -3.81, -1193.545]
  MoveL 489 to (21.11, 178.51, 150) mm, rotated rx -90 ry -25 rz 66.45 deg; joints [-1.904, -48.989, 102.686, 37.787, -108.022, -3.536, -1186.447]
  MoveL 490 to (11.96, 176.54, 140) mm, rotated rx -90 ry -25 rz 59.25 deg; joints [-2.265, -49.133, 102.976, 37.58, -108.007, -3.265, -1179.249]
  MoveL 491 to (2.59, 175.67, 130) mm, rotated rx -90 ry -25 rz 51.99 deg; joints [-2.628, -49.278, 103.259, 37.369, -107.986, -2.998, -1171.995]
  MoveL 492 to (-6.83, 175.92, 120) mm, rotated rx -90 ry -25 rz 44.73 deg; joints [-2.992, -49.422, 103.535, 37.155, -107.962, -2.735, -1164.728]
  MoveL 493 to (-16.13, 177.3, 110) mm, rotated rx -90 ry -25 rz 37.49 deg; joints [-3.358, -49.566, 103.804, 36.938, -107.933, -2.476, -1157.494]
  MoveL 494 to (-25.11, 179.73, 100) mm, rotated rx -90 ry -25 rz 30.34 deg; joints [-3.725, -49.71, 104.067, 36.719, -107.9, -2.221, -1150.336]
  MoveL 495 to (-33.62, 183.16, 90) mm, rotated rx -90 ry -25 rz 23.3 deg; joints [-4.093, -49.853, 104.323, 36.496, -107.862, -1.969, -1143.298]
  MoveL 496 to (-41.52, 187.45, 80) mm, rotated rx -90 ry -25 rz 16.42 deg; joints [-4.463, -49.996, 104.573, 36.271, -107.821, -1.721, -1136.42]
  MoveL 497 to (-48.7, 192.48, 70) mm, rotated rx -90 ry -25 rz 9.74 deg; joints [-4.834, -50.138, 104.816, 36.043, -107.777, -1.476, -1129.745]
  MoveL 498 to (-55.08, 198.08, 60) mm, rotated rx -90 ry -25 rz 3.31 deg; joints [-5.207, -50.278, 105.053, 35.813, -107.729, -1.233, -1123.31]
  MoveL 499 to (-60.61, 204.07, 50) mm, rotated rx -90 ry -25 rz -2.85 deg; joints [-5.581, -50.415, 105.283, 35.581, -107.678, -0.993, -1117.152]
  MoveL 500 to (-65.29, 210.3, 40) mm, rotated rx -90 ry -25 rz -8.69 deg; joints [-5.956, -50.551, 105.507, 35.346, -107.625, -0.755, -1111.307]
  MoveL 501 to (-69.12, 216.58, 30) mm, rotated rx -90 ry -25 rz -14.19 deg; joints [-6.332, -50.683, 105.725, 35.11, -107.571, -0.518, -1105.808]
  MoveL 502 to (-72.16, 222.75, 20) mm, rotated rx -90 ry -25 rz -19.31 deg; joints [-6.709, -50.811, 105.937, 34.871, -107.515, -0.282, -1100.687]
  MoveL 503 to (-74.48, 228.68, 10) mm, rotated rx -90 ry -25 rz -24.02 deg; joints [-7.088, -50.936, 106.142, 34.631, -107.458, -0.048, -1095.978]
  MoveL 504 to (-76.17, 234.21, 0) mm, rotated rx -90 ry -25 rz -28.29 deg; joints [-7.468, -51.057, 106.341, 34.389, -107.4, 0.186, -1091.709]
  Set speed (1000.0 mm/s)
  MoveL 505 to (-76.17, 234.21, 0) mm, rotated rx -90 ry -25 rz -28.29 deg; joints [-7.468, -51.057, 106.341, 34.389, -107.4, 0.186, -1091.709]
  Set speed (1000.0 mm/s)
  MoveL 506 to (78.63, 249.2, 290) mm, rotated rx -90 ry -25 rz 139.42 deg; joints [2.992, -46.728, 97.946, 40.411, -107.981, -7.612, -1259.419]
  MoveL 507 to (78.63, 249.2, 290) mm, rotated rx -90 ry -25 rz 139.42 deg; joints [2.992, -46.728, 97.946, 40.411, -107.981, -7.612, -1259.419]
  Set speed (60.0 mm/s)
  MoveL 508 to (58.93, 255.88, 290) mm, rotated rx -90 ry -25 rz 145.69 deg; joints [2.992, -45.858, 98.042, 40.619, -108.716, -6.951, -1265.694]
  Set speed (1000.0 mm/s)
  MoveL 509 to (58.93, 255.88, 290) mm, rotated rx -90 ry -25 rz 145.69 deg; joints [2.992, -45.858, 98.042, 40.619, -108.716, -6.951, -1265.694]
  Set speed (1000.0 mm/s)
  MoveL 510 to (-76.17, 234.21, 0) mm, rotated rx -90 ry -25 rz -28.29 deg; joints [-7.468, -51.057, 106.341, 34.389, -107.4, 0.186, -1091.709]
  MoveL 511 to (-76.17, 234.21, 0) mm, rotated rx -90 ry -25 rz -28.29 deg; joints [-7.468, -51.057, 106.341, 34.389, -107.4, 0.186, -1091.709]
  Set speed (60.0 mm/s)
  MoveL 512 to (-55.37, 234.2, 0) mm, rotated rx -90 ry -25 rz -24.07 deg; joints [-7.468, -50.074, 106.439, 34.586, -108.291, 0.829, -1095.929]
  Set speed (1000.0 mm/s)
  MoveL 513 to (-55.37, 234.2, 0) mm, rotated rx -90 ry -25 rz -24.07 deg; joints [-7.468, -50.074, 106.439, 34.586, -108.291, 0.829, -1095.929]
  Set speed (1000.0 mm/s)
  MoveL 514 to (-76.17, 234.21, 0) mm, rotated rx -90 ry -25 rz -28.29 deg; joints [-7.468, -51.057, 106.341, 34.389, -107.4, 0.186, -1091.709]
  MoveL 515 to (-76.17, 234.21, 0) mm, rotated rx -90 ry -25 rz -28.29 deg; joints [-7.468, -51.057, 106.341, 34.389, -107.4, 0.186, -1091.709]
  Set speed (60.0 mm/s)
  MoveL 516 to (-74.48, 228.68, 10) mm, rotated rx -90 ry -25 rz -24.02 deg; joints [-7.088, -50.936, 106.142, 34.631, -107.458, -0.048, -1095.978]
  MoveL 517 to (-72.16, 222.75, 20) mm, rotated rx -90 ry -25 rz -19.31 deg; joints [-6.709, -50.811, 105.937, 34.871, -107.515, -0.282, -1100.687]
  MoveL 518 to (-69.12, 216.58, 30) mm, rotated rx -90 ry -25 rz -14.19 deg; joints [-6.332, -50.683, 105.725, 35.11, -107.571, -0.518, -1105.808]
  MoveL 519 to (-65.29, 210.3, 40) mm, rotated rx -90 ry -25 rz -8.69 deg; joints [-5.956, -50.551, 105.507, 35.346, -107.625, -0.755, -1111.307]
  MoveL 520 to (-60.61, 204.07, 50) mm, rotated rx -90 ry -25 rz -2.85 deg; joints [-5.581, -50.415, 105.283, 35.581, -107.678, -0.993, -1117.152]
  MoveL 521 to (-55.08, 198.08, 60) mm, rotated rx -90 ry -25 rz 3.31 deg; joints [-5.207, -50.278, 105.053, 35.813, -107.729, -1.233, -1123.31]
  MoveL 522 to (-48.7, 192.48, 70) mm, rotated rx -90 ry -25 rz 9.74 deg; joints [-4.834, -50.138, 104.816, 36.043, -107.777, -1.476, -1129.745]
  MoveL 523 to (-41.52, 187.45, 80) mm, rotated rx -90 ry -25 rz 16.42 deg; joints [-4.463, -49.996, 104.573, 36.271, -107.821, -1.721, -1136.42]
  MoveL 524 to (-33.62, 183.16, 90) mm, rotated rx -90 ry -25 rz 23.3 deg; joints [-4.093, -49.853, 104.323, 36.496, -107.862, -1.969, -1143.298]
  MoveL 525 to (-25.11, 179.73, 100) mm, rotated rx -90 ry -25 rz 30.34 deg; joints [-3.725, -49.71, 104.067, 36.719, -107.9, -2.221, -1150.336]
  MoveL 526 to (-16.13, 177.3, 110) mm, rotated rx -90 ry -25 rz 37.49 deg; joints [-3.358, -49.566, 103.804, 36.938, -107.933, -2.476, -1157.494]
  MoveL 527 to (-6.83, 175.92, 120) mm, rotated rx -90 ry -25 rz 44.73 deg; joints [-2.992, -49.422, 103.535, 37.155, -107.962, -2.735, -1164.728]
  MoveL 528 to (2.59, 175.67, 130) mm, rotated rx -90 ry -25 rz 51.99 deg; joints [-2.628, -49.278, 103.259, 37.369, -107.986, -2.998, -1171.995]
  MoveL 529 to (11.96, 176.54, 140) mm, rotated rx -90 ry -25 rz 59.25 deg; joints [-2.265, -49.133, 102.976, 37.58, -108.007, -3.265, -1179.249]
  MoveL 530 to (21.11, 178.51, 150) mm, rotated rx -90 ry -25 rz 66.45 deg; joints [-1.904, -48.989, 102.686, 37.787, -108.022, -3.536, -1186.447]
  MoveL 531 to (29.85, 181.5, 160) mm, rotated rx -90 ry -25 rz 73.54 deg; joints [-1.544, -48.844, 102.39, 37.992, -108.034, -3.81, -1193.545]
  MoveL 532 to (38.04, 185.42, 170) mm, rotated rx -90 ry -25 rz 80.5 deg; joints [-1.185, -48.698, 102.087, 38.194, -108.042, -4.089, -1200.5]
  MoveL 533 to (45.56, 190.13, 180) mm, rotated rx -90 ry -25 rz 87.27 deg; joints [-0.828, -48.551, 101.778, 38.393, -108.047, -4.371, -1207.271]
  MoveL 534 to (52.31, 195.49, 190) mm, rotated rx -90 ry -25 rz 93.82 deg; joints [-0.473, -48.403, 101.462, 38.589, -108.049, -4.656, -1213.819]
  MoveL 535 to (58.22, 201.33, 200) mm, rotated rx -90 ry -25 rz 100.11 deg; joints [-0.119, -48.252, 101.139, 38.782, -108.048, -4.944, -1220.107]
  MoveL 536 to (63.28, 207.47, 210) mm, rotated rx -90 ry -25 rz 106.1 deg; joints [0.233, -48.099, 100.81, 38.972, -108.044, -5.234, -1226.097]
  MoveL 537 to (67.49, 213.75, 220) mm, rotated rx -90 ry -25 rz 111.76 deg; joints [0.584, -47.942, 100.475, 39.16, -108.039, -5.526, -1231.756]
  MoveL 538 to (70.88, 219.99, 230) mm, rotated rx -90 ry -25 rz 117.05 deg; joints [0.933, -47.782, 100.133, 39.346, -108.033, -5.821, -1237.052]
  MoveL 539 to (73.51, 226.04, 240) mm, rotated rx -90 ry -25 rz 121.95 deg; joints [1.28, -47.618, 99.784, 39.529, -108.026, -6.117, -1241.95]
  MoveL 540 to (75.48, 231.77, 250) mm, rotated rx -90 ry -25 rz 126.42 deg; joints [1.626, -47.45, 99.43, 39.71, -108.018, -6.414, -1246.422]
  MoveL 541 to (76.86, 237.05, 260) mm, rotated rx -90 ry -25 rz 130.43 deg; joints [1.97, -47.277, 99.068, 39.888, -108.009, -6.712, -1250.435]
  MoveL 542 to (77.78, 241.77, 270) mm, rotated rx -90 ry -25 rz 133.96 deg; joints [2.312, -47.099, 98.701, 40.065, -108, -7.012, -1253.959]
  MoveL 543 to (78.34, 245.85, 280) mm, rotated rx -90 ry -25 rz 136.96 deg; joints [2.653, -46.916, 98.327, 40.239, -107.991, -7.312, -1256.964]
  MoveL 544 to (78.63, 249.2, 290) mm, rotated rx -90 ry -25 rz 139.42 deg; joints [2.992, -46.728, 97.946, 40.411, -107.981, -7.612, -1259.419]
  Set speed (1000.0 mm/s)
  MoveL 545 to (78.63, 249.2, 290) mm, rotated rx -90 ry -25 rz 139.42 deg; joints [2.992, -46.728, 97.946, 40.411, -107.981, -7.612, -1259.419]
  Set speed (1000.0 mm/s)
  MoveL 546 to (58.93, 255.88, 290) mm, rotated rx -90 ry -25 rz 145.69 deg; joints [2.992, -45.858, 98.042, 40.619, -108.716, -6.951, -1265.694]
  MoveL 547 to (58.93, 255.88, 290) mm, rotated rx -90 ry -25 rz 145.69 deg; joints [2.992, -45.858, 98.042, 40.619, -108.716, -6.951, -1265.694]
  Set speed (60.0 mm/s)
  MoveL 548 to (58.94, 253.36, 280) mm, rotated rx -90 ry -25 rz 143.26 deg; joints [2.653, -46.043, 98.422, 40.447, -108.729, -6.651, -1263.258]
  MoveL 549 to (58.8, 250.28, 270) mm, rotated rx -90 ry -25 rz 140.27 deg; joints [2.312, -46.222, 98.796, 40.273, -108.742, -6.351, -1260.274]
  MoveL 550 to (58.44, 246.7, 260) mm, rotated rx -90 ry -25 rz 136.77 deg; joints [1.97, -46.397, 99.163, 40.097, -108.755, -6.052, -1256.77]
  MoveL 551 to (57.77, 242.68, 250) mm, rotated rx -90 ry -25 rz 132.77 deg; joints [1.626, -46.567, 99.524, 39.918, -108.768, -5.755, -1252.774]
  MoveL 552 to (56.69, 238.28, 240) mm, rotated rx -90 ry -25 rz 128.32 deg; joints [1.28, -46.731, 99.878, 39.737, -108.781, -5.458, -1248.316]
  MoveL 553 to (55.14, 233.59, 230) mm, rotated rx -90 ry -25 rz 123.42 deg; joints [0.933, -46.892, 100.226, 39.554, -108.793, -5.162, -1243.424]
  MoveL 554 to (53.04, 228.71, 220) mm, rotated rx -90 ry -25 rz 118.13 deg; joints [0.584, -47.048, 100.567, 39.369, -108.804, -4.868, -1238.126]
  MoveL 555 to (50.33, 223.75, 210) mm, rotated rx -90 ry -25 rz 112.45 deg; joints [0.233, -47.2, 100.902, 39.181, -108.813, -4.576, -1232.453]
  MoveL 556 to (46.98, 218.83, 200) mm, rotated rx -90 ry -25 rz 106.43 deg; joints [-0.119, -47.349, 101.231, 38.99, -108.822, -4.286, -1226.434]
  MoveL 557 to (42.97, 214.08, 190) mm, rotated rx -90 ry -25 rz 100.1 deg; joints [-0.473, -47.495, 101.553, 38.797, -108.828, -3.998, -1220.103]
  MoveL 558 to (38.31, 209.62, 180) mm, rotated rx -90 ry -25 rz 93.49 deg; joints [-0.828, -47.639, 101.869, 38.601, -108.832, -3.713, -1213.494]
  MoveL 559 to (33.03, 205.6, 170) mm, rotated rx -90 ry -25 rz 86.64 deg; joints [-1.185, -47.781, 102.178, 38.402, -108.833, -3.431, -1206.645]
  MoveL 560 to (27.19, 202.13, 160) mm, rotated rx -90 ry -25 rz 79.59 deg; joints [-1.544, -47.922, 102.481, 38.2, -108.831, -3.152, -1199.594]
  MoveL 561 to (20.88, 199.3, 150) mm, rotated rx -90 ry -25 rz 72.38 deg; joints [-1.904, -48.062, 102.777, 37.995, -108.826, -2.877, -1192.384]
  MoveL 562 to (14.2, 197.22, 140) mm, rotated rx -90 ry -25 rz 65.06 deg; joints [-2.265, -48.201, 103.066, 37.788, -108.816, -2.606, -1185.059]
  MoveL 563 to (7.28, 195.93, 130) mm, rotated rx -90 ry -25 rz 57.67 deg; joints [-2.628, -48.34, 103.349, 37.577, -108.802, -2.339, -1177.666]
  MoveL 564 to (0.24, 195.48, 120) mm, rotated rx -90 ry -25 rz 50.25 deg; joints [-2.992, -48.479, 103.625, 37.363, -108.784, -2.076, -1170.252]
  MoveL 565 to (-6.77, 195.87, 110) mm, rotated rx -90 ry -25 rz 42.87 deg; joints [-3.358, -48.619, 103.895, 37.146, -108.762, -1.817, -1162.866]
  MoveL 566 to (-13.63, 197.08, 100) mm, rotated rx -90 ry -25 rz 35.55 deg; joints [-3.725, -48.758, 104.159, 36.926, -108.735, -1.562, -1155.555]
  MoveL 567 to (-20.21, 199.05, 90) mm, rotated rx -90 ry -25 rz 28.37 deg; joints [-4.093, -48.897, 104.415, 36.703, -108.704, -1.311, -1148.366]
  MoveL 568 to (-26.38, 201.72, 80) mm, rotated rx -90 ry -25 rz 21.35 deg; joints [-4.463, -49.036, 104.666, 36.477, -108.669, -1.064, -1141.346]
  MoveL 569 to (-32.08, 204.97, 70) mm, rotated rx -90 ry -25 rz 14.54 deg; joints [-4.834, -49.174, 104.909, 36.248, -108.63, -0.819, -1134.536]
  MoveL 570 to (-37.21, 208.71, 60) mm, rotated rx -90 ry -25 rz 7.98 deg; joints [-5.207, -49.31, 105.147, 36.017, -108.588, -0.578, -1127.979]
  MoveL 571 to (-41.73, 212.8, 50) mm, rotated rx -90 ry -25 rz 1.71 deg; joints [-5.581, -49.445, 105.378, 35.784, -108.543, -0.339, -1121.712]
  MoveL 572 to (-45.64, 217.12, 40) mm, rotated rx -90 ry -25 rz -4.23 deg; joints [-5.956, -49.577, 105.603, 35.548, -108.496, -0.103, -1115.772]
  MoveL 573 to (-48.92, 221.54, 30) mm, rotated rx -90 ry -25 rz -9.81 deg; joints [-6.332, -49.707, 105.821, 35.31, -108.447, 0.132, -1110.192]
  MoveL 574 to (-51.6, 225.93, 20) mm, rotated rx -90 ry -25 rz -15 deg; joints [-6.709, -49.833, 106.033, 35.071, -108.396, 0.365, -1105.005]
  MoveL 575 to (-53.73, 230.19, 10) mm, rotated rx -90 ry -25 rz -19.76 deg; joints [-7.088, -49.956, 106.239, 34.829, -108.344, 0.598, -1100.24]
  MoveL 576 to (-55.37, 234.2, 0) mm, rotated rx -90 ry -25 rz -24.07 deg; joints [-7.468, -50.074, 106.439, 34.586, -108.291, 0.829, -1095.929]
  Set speed (1000.0 mm/s)
  MoveL 577 to (-55.37, 234.2, 0) mm, rotated rx -90 ry -25 rz -24.07 deg; joints [-7.468, -50.074, 106.439, 34.586, -108.291, 0.829, -1095.929]
  Set speed (1000.0 mm/s)
  MoveL 578 to (58.93, 255.88, 290) mm, rotated rx -90 ry -25 rz 145.69 deg; joints [2.992, -45.858, 98.042, 40.619, -108.716, -6.951, -1265.694]
  MoveL 579 to (58.93, 255.88, 290) mm, rotated rx -90 ry -25 rz 145.69 deg; joints [2.992, -45.858, 98.042, 40.619, -108.716, -6.951, -1265.694]
  Set speed (60.0 mm/s)
  MoveL 580 to (37.11, 300.24, 290) mm, rotated rx -90 ry -25 rz -166.45 deg; joints [2.992, -46.004, 98.028, 40.584, -108.594, -7.061, -1313.547]
  Set speed (1000.0 mm/s)
  MoveL 581 to (37.11, 300.24, 290) mm, rotated rx -90 ry -25 rz -166.45 deg; joints [2.992, -46.004, 98.028, 40.584, -108.594, -7.061, -1313.547]
  Set speed (1000.0 mm/s)
  MoveL 582 to (-55.37, 234.2, 0) mm, rotated rx -90 ry -25 rz -24.07 deg; joints [-7.468, -50.074, 106.439, 34.586, -108.291, 0.829, -1455.929]
  MoveL 583 to (-55.37, 234.2, 0) mm, rotated rx -90 ry -25 rz -24.07 deg; joints [-7.468, -50.074, 106.439, 34.586, -108.291, 0.829, -1455.929]
  Set speed (60.0 mm/s)
  MoveL 584 to (-20.49, 199.16, 0) mm, rotated rx -90 ry -25 rz 28.05 deg; joints [-7.468, -49.938, 106.45, 34.613, -108.412, 0.917, -1508.047]
  Set speed (1000.0 mm/s)
  MoveL 585 to (-20.49, 199.16, 0) mm, rotated rx -90 ry -25 rz 28.05 deg; joints [-7.468, -49.938, 106.45, 34.613, -108.412, 0.917, -1508.047]
  Set speed (1000.0 mm/s)
  MoveL 586 to (-55.37, 234.2, 0) mm, rotated rx -90 ry -25 rz -24.07 deg; joints [-7.468, -50.074, 106.439, 34.586, -108.291, 0.829, -1455.929]
  MoveL 587 to (-55.37, 234.2, 0) mm, rotated rx -90 ry -25 rz -24.07 deg; joints [-7.468, -50.074, 106.439, 34.586, -108.291, 0.829, -1455.929]
  Set speed (60.0 mm/s)
  MoveL 588 to (-53.73, 230.19, 10) mm, rotated rx -90 ry -25 rz -19.76 deg; joints [-7.088, -49.956, 106.239, 34.829, -108.344, 0.598, -1460.24]
  MoveL 589 to (-51.6, 225.93, 20) mm, rotated rx -90 ry -25 rz -15 deg; joints [-6.709, -49.833, 106.033, 35.071, -108.396, 0.365, -1465.005]
  MoveL 590 to (-48.92, 221.54, 30) mm, rotated rx -90 ry -25 rz -9.81 deg; joints [-6.332, -49.707, 105.821, 35.31, -108.447, 0.132, -1470.192]
  MoveL 591 to (-45.64, 217.12, 40) mm, rotated rx -90 ry -25 rz -4.23 deg; joints [-5.956, -49.577, 105.603, 35.548, -108.496, -0.103, -1475.772]
  MoveL 592 to (-41.73, 212.8, 50) mm, rotated rx -90 ry -25 rz 1.71 deg; joints [-5.581, -49.445, 105.378, 35.784, -108.543, -0.339, -1481.712]
  MoveL 593 to (-37.21, 208.71, 60) mm, rotated rx -90 ry -25 rz 7.98 deg; joints [-5.207, -49.31, 105.147, 36.017, -108.588, -0.578, -1487.979]
  MoveL 594 to (-32.08, 204.97, 70) mm, rotated rx -90 ry -25 rz 14.54 deg; joints [-4.834, -49.174, 104.909, 36.248, -108.63, -0.819, -1494.536]
  MoveL 595 to (-26.38, 201.72, 80) mm, rotated rx -90 ry -25 rz 21.35 deg; joints [-4.463, -49.036, 104.666, 36.477, -108.669, -1.064, -1501.346]
  MoveL 596 to (-20.21, 199.05, 90) mm, rotated rx -90 ry -25 rz 28.37 deg; joints [-4.093, -48.897, 104.415, 36.703, -108.704, -1.311, -1508.366]
  MoveL 597 to (-13.63, 197.08, 100) mm, rotated rx -90 ry -25 rz 35.55 deg; joints [-3.725, -48.758, 104.159, 36.926, -108.735, -1.562, -1515.555]
  MoveL 598 to (-6.77, 195.87, 110) mm, rotated rx -90 ry -25 rz 42.87 deg; joints [-3.358, -48.619, 103.895, 37.146, -108.762, -1.817, -1522.866]
  MoveL 599 to (0.24, 195.48, 120) mm, rotated rx -90 ry -25 rz 50.25 deg; joints [-2.992, -48.479, 103.625, 37.363, -108.784, -2.076, -1530.252]
  MoveL 600 to (7.28, 195.93, 130) mm, rotated rx -90 ry -25 rz 57.67 deg; joints [-2.628, -48.34, 103.349, 37.577, -108.802, -2.339, -1537.666]
  MoveL 601 to (14.2, 197.22, 140) mm, rotated rx -90 ry -25 rz 65.06 deg; joints [-2.265, -48.201, 103.066, 37.788, -108.816, -2.606, -1545.059]
  MoveL 602 to (20.88, 199.3, 150) mm, rotated rx -90 ry -25 rz 72.38 deg; joints [-1.904, -48.062, 102.777, 37.995, -108.826, -2.877, -1552.384]
  MoveL 603 to (27.19, 202.13, 160) mm, rotated rx -90 ry -25 rz 79.59 deg; joints [-1.544, -47.922, 102.481, 38.2, -108.831, -3.152, -1559.594]
  MoveL 604 to (33.03, 205.6, 170) mm, rotated rx -90 ry -25 rz 86.64 deg; joints [-1.185, -47.781, 102.178, 38.402, -108.833, -3.431, -1566.645]
  MoveL 605 to (38.31, 209.62, 180) mm, rotated rx -90 ry -25 rz 93.49 deg; joints [-0.828, -47.639, 101.869, 38.601, -108.832, -3.713, -1573.494]
  MoveL 606 to (42.97, 214.08, 190) mm, rotated rx -90 ry -25 rz 100.1 deg; joints [-0.473, -47.495, 101.553, 38.797, -108.828, -3.998, -1580.103]
  MoveL 607 to (46.98, 218.83, 200) mm, rotated rx -90 ry -25 rz 106.43 deg; joints [-0.119, -47.349, 101.231, 38.99, -108.822, -4.286, -1586.434]
  MoveL 608 to (50.33, 223.75, 210) mm, rotated rx -90 ry -25 rz 112.45 deg; joints [0.233, -47.2, 100.902, 39.181, -108.813, -4.576, -1592.453]
  MoveL 609 to (53.04, 228.71, 220) mm, rotated rx -90 ry -25 rz 118.13 deg; joints [0.584, -47.048, 100.567, 39.369, -108.804, -4.868, -1598.126]
  MoveL 610 to (55.14, 233.59, 230) mm, rotated rx -90 ry -25 rz 123.42 deg; joints [0.933, -46.892, 100.226, 39.554, -108.793, -5.162, -1603.424]
  MoveL 611 to (56.69, 238.28, 240) mm, rotated rx -90 ry -25 rz 128.32 deg; joints [1.28, -46.731, 99.878, 39.737, -108.781, -5.458, -1608.316]
  MoveL 612 to (57.77, 242.68, 250) mm, rotated rx -90 ry -25 rz 132.77 deg; joints [1.626, -46.567, 99.524, 39.918, -108.768, -5.755, -1612.774]
  MoveL 613 to (58.44, 246.7, 260) mm, rotated rx -90 ry -25 rz 136.77 deg; joints [1.97, -46.397, 99.163, 40.097, -108.755, -6.052, -1616.77]
  MoveL 614 to (58.8, 250.28, 270) mm, rotated rx -90 ry -25 rz 140.27 deg; joints [2.312, -46.222, 98.796, 40.273, -108.742, -6.351, -1620.274]
  MoveL 615 to (58.94, 253.36, 280) mm, rotated rx -90 ry -25 rz 143.26 deg; joints [2.653, -46.043, 98.422, 40.447, -108.729, -6.651, -1623.258]
  MoveL 616 to (58.93, 255.88, 290) mm, rotated rx -90 ry -25 rz 145.69 deg; joints [2.992, -45.858, 98.042, 40.619, -108.716, -6.951, -1625.694]
  Set speed (1000.0 mm/s)
  MoveL 617 to (58.93, 255.88, 290) mm, rotated rx -90 ry -25 rz 145.69 deg; joints [2.992, -45.858, 98.042, 40.619, -108.716, -6.951, -1625.694]
  Set speed (1000.0 mm/s)
  MoveL 618 to (37.11, 300.24, 290) mm, rotated rx -96.9 ry -17.88 rz 75.79 deg; joints [-1.762, -22.307, 19.15, 141.67, -56.455, -149.47, -1646.629]
  MoveL 619 to (37.11, 300.24, 290) mm, rotated rx -96.9 ry -17.88 rz 75.79 deg; joints [-1.762, -22.307, 19.15, 141.67, -56.455, -149.47, -1646.629]
  Set speed (60.0 mm/s)
  MoveL 620 to (39.03, 298.61, 280) mm, rotated rx -97.08 ry -15.54 rz 79.68 deg; joints [-1.817, -34.316, 42.197, 131.116, -41.994, -135.035, -1643.609]
  MoveL 621 to (41.29, 296.51, 270) mm, rotated rx -98.79 ry -14.56 rz 73.06 deg; joints [-2.194, -31.58, 37.029, 137.372, -44.628, -143.492, -1640.035]
  MoveL 622 to (43.78, 293.91, 260) mm, rotated rx -100.6 ry -13.96 rz 65.48 deg; joints [-2.524, -27.364, 29.096, 143.507, -49.428, -152.28, -1635.959]
  MoveL 623 to (44.93, 293.38, 249.12) mm, rotated rx -102.48 ry -13.76 rz 57.03 deg; joints [-2.804, -17.515, 10.028, 150.069, -60.063, -163.189, -1631.425]
  MoveL 624 to (49.06, 287.12, 240) mm, rotated rx -75.01 ry -14.65 rz 147.83 deg; joints [-3.224, -48.207, 108.443, 27.099, -113.884, 12.342, -1626.478]
  MoveL 625 to (51.62, 282.9, 230) mm, rotated rx -75.3 ry -12.71 rz 137.52 deg; joints [-3.935, -50.762, 109.257, 24.608, -107.196, 9.803, -1621.161]
  MoveL 626 to (53.98, 278.14, 220) mm, rotated rx -73.63 ry -13.16 rz 135.62 deg; joints [-4.597, -49.036, 109.478, 24.655, -112.497, 13.57, -1615.515]
  MoveL 627 to (56, 272.86, 210) mm, rotated rx -72.12 ry -13.76 rz 133.16 deg; joints [-5.21, -47.279, 109.363, 25.11, -117.258, 17.177, -1609.582]
  MoveL 628 to (57.57, 267.12, 200) mm, rotated rx -73 ry -11.66 rz 121.38 deg; joints [-5.837, -50.269, 110.344, 22.253, -109.766, 13.657, -1603.4]
  MoveL 629 to (58.59, 260.98, 190) mm, rotated rx -71.71 ry -12.29 rz 118.09 deg; joints [-6.387, -48.731, 110.34, 22.647, -114.135, 16.697, -1597.009]
  MoveL 630 to (58.95, 254.55, 180) mm, rotated rx -70.55 ry -13.02 rz 114.47 deg; joints [-6.895, -47.173, 110.109, 23.335, -118.142, 19.663, -1590.447]
  MoveL 631 to (58.59, 247.92, 170) mm, rotated rx -71.88 ry -10.84 rz 101.84 deg; joints [-7.456, -50.401, 111.102, 20.323, -110.121, 15.539, -1583.752]
  MoveL 632 to (57.45, 241.22, 160) mm, rotated rx -70.86 ry -11.6 rz 97.82 deg; joints [-7.918, -48.992, 111.026, 20.911, -114.028, 18.097, -1576.959]
  MoveL 633 to (55.51, 234.59, 150) mm, rotated rx -69.95 ry -12.44 rz 93.68 deg; joints [-8.342, -47.538, 110.762, 21.759, -117.727, 20.659, -1570.107]
  MoveL 634 to (52.77, 228.15, 140) mm, rotated rx -71.59 ry -10.32 rz 80.79 deg; joints [-8.837, -50.822, 111.649, 18.83, -109.469, 16.265, -1563.231]
  MoveL 635 to (49.26, 222.05, 130) mm, rotated rx -70.76 ry -11.22 rz 76.66 deg; joints [-9.222, -49.431, 111.542, 19.623, -113.329, 18.576, -1556.367]
